  PROC DrawPart60()
    MoveL Offs(pOrigin,354.34,117.20,0.00),v40,z0,tPen\WObj:=wPaper;
    MoveL Offs(pOrigin,355.40,117.41,0.00),v40,z0,tPen\WObj:=wPaper;
    MoveL Offs(pOrigin,355.40,117.41,0.00),v40,z0,tPen\WObj:=wPaper;
    MoveL Offs(pOrigin,357.74,120.39,0.00),v40,z0,tPen\WObj:=wPaper;
    MoveL Offs(pOrigin,361.56,124.00,0.00),v40,z0,tPen\WObj:=wPaper;
    MoveL Offs(pOrigin,364.33,126.12,0.00),v40,z0,tPen\WObj:=wPaper;
    MoveL Offs(pOrigin,368.79,128.89,0.00),v40,fine,tPen\WObj:=wPaper;
    MoveL Offs(pOrigin,368.79,128.89,6.00),v60,z5,tPen\WObj:=wPaper;
    MoveL Offs(pOrigin,367.20,127.37,6.00),vTravel,z5,tPen\WObj:=wPaper;
    MoveL Offs(pOrigin,367.20,127.37,0.00),v60,z0,tPen\WObj:=wPaper;
    MoveL Offs(pOrigin,366.30,128.27,0.00),v40,z0,tPen\WObj:=wPaper;
    MoveL Offs(pOrigin,365.40,127.67,0.00),v40,z0,tPen\WObj:=wPaper;
    MoveL Offs(pOrigin,366.30,126.77,0.00),v40,z0,tPen\WObj:=wPaper;
    MoveL Offs(pOrigin,365.56,126.02,0.00),v40,z0,tPen\WObj:=wPaper;
    MoveL Offs(pOrigin,364.51,127.07,0.00),v40,z0,tPen\WObj:=wPaper;
    MoveL Offs(pOrigin,363.46,126.63,0.00),v40,z0,tPen\WObj:=wPaper;
    MoveL Offs(pOrigin,364.81,125.28,0.00),v40,z0,tPen\WObj:=wPaper;
    MoveL Offs(pOrigin,364.06,124.53,0.00),v40,z0,tPen\WObj:=wPaper;
    MoveL Offs(pOrigin,362.56,126.03,0.00),v40,fine,tPen\WObj:=wPaper;
    MoveL Offs(pOrigin,362.56,126.03,6.00),v60,z5,tPen\WObj:=wPaper;
    MoveL Offs(pOrigin,358.96,129.64,6.00),vTravel,z5,tPen\WObj:=wPaper;
    MoveL Offs(pOrigin,358.96,129.64,0.00),v60,z0,tPen\WObj:=wPaper;
    MoveL Offs(pOrigin,352.19,136.40,0.00),v40,z0,tPen\WObj:=wPaper;
    MoveL Offs(pOrigin,352.71,136.45,0.00),v40,z0,tPen\WObj:=wPaper;
    MoveL Offs(pOrigin,355.71,139.46,0.00),v40,z0,tPen\WObj:=wPaper;
    MoveL Offs(pOrigin,355.40,139.61,0.00),v40,z0,tPen\WObj:=wPaper;
    MoveL Offs(pOrigin,354.12,139.61,0.00),v40,z0,tPen\WObj:=wPaper;
    MoveL Offs(pOrigin,353.77,140.50,0.00),v40,z0,tPen\WObj:=wPaper;
    MoveL Offs(pOrigin,356.62,143.36,0.00),v40,z0,tPen\WObj:=wPaper;
    MoveL Offs(pOrigin,356.46,143.83,0.00),v40,z0,tPen\WObj:=wPaper;
    MoveL Offs(pOrigin,355.19,143.83,0.00),v40,z0,tPen\WObj:=wPaper;
    MoveL Offs(pOrigin,354.68,144.40,0.00),v40,z0,tPen\WObj:=wPaper;
    MoveL Offs(pOrigin,357.68,147.41,0.00),v40,z0,tPen\WObj:=wPaper;
    MoveL Offs(pOrigin,358.00,147.02,0.00),v40,z0,tPen\WObj:=wPaper;
    MoveL Offs(pOrigin,355.60,149.42,0.00),v40,z0,tPen\WObj:=wPaper;
    MoveL Offs(pOrigin,356.46,149.11,0.00),v40,z0,tPen\WObj:=wPaper;
    MoveL Offs(pOrigin,357.52,149.11,0.00),v40,z0,tPen\WObj:=wPaper;
    MoveL Offs(pOrigin,358.14,149.35,0.00),v40,z0,tPen\WObj:=wPaper;
    MoveL Offs(pOrigin,355.13,146.35,0.00),v40,z0,tPen\WObj:=wPaper;
    MoveL Offs(pOrigin,355.61,145.94,0.00),v40,z0,tPen\WObj:=wPaper;
    MoveL Offs(pOrigin,356.89,145.94,0.00),v40,z0,tPen\WObj:=wPaper;
    MoveL Offs(pOrigin,357.23,145.46,0.00),v40,z0,tPen\WObj:=wPaper;
    MoveL Offs(pOrigin,354.22,142.45,0.00),v40,z0,tPen\WObj:=wPaper;
    MoveL Offs(pOrigin,353.82,142.24,0.00),v40,z0,tPen\WObj:=wPaper;
    MoveL Offs(pOrigin,356.38,139.68,0.00),v40,fine,tPen\WObj:=wPaper;
    MoveL Offs(pOrigin,356.38,139.68,6.00),v60,z5,tPen\WObj:=wPaper;
    MoveL Offs(pOrigin,356.08,138.49,6.00),vTravel,z5,tPen\WObj:=wPaper;
    MoveL Offs(pOrigin,356.08,138.49,0.00),v60,z0,tPen\WObj:=wPaper;
    MoveL Offs(pOrigin,353.53,141.04,0.00),v40,z0,tPen\WObj:=wPaper;
    MoveL Offs(pOrigin,354.34,140.66,0.00),v40,z0,tPen\WObj:=wPaper;
    MoveL Offs(pOrigin,355.61,140.66,0.00),v40,z0,tPen\WObj:=wPaper;
    MoveL Offs(pOrigin,356.17,141.41,0.00),v40,z0,tPen\WObj:=wPaper;
    MoveL Offs(pOrigin,353.16,138.40,0.00),v40,z0,tPen\WObj:=wPaper;
    MoveL Offs(pOrigin,352.94,138.64,0.00),v40,z0,tPen\WObj:=wPaper;
    MoveL Offs(pOrigin,360.30,131.28,0.00),v40,z0,tPen\WObj:=wPaper;
    MoveL Offs(pOrigin,360.08,132.22,0.00),v40,z0,tPen\WObj:=wPaper;
    MoveL Offs(pOrigin,358.16,132.22,0.00),v40,fine,tPen\WObj:=wPaper;
    MoveL Offs(pOrigin,358.16,132.22,6.00),v60,z5,tPen\WObj:=wPaper;
    MoveL Offs(pOrigin,359.23,131.44,6.00),vTravel,z5,tPen\WObj:=wPaper;
    MoveL Offs(pOrigin,359.23,131.44,0.00),v60,z0,tPen\WObj:=wPaper;
    MoveL Offs(pOrigin,359.65,131.86,0.00),v40,z0,tPen\WObj:=wPaper;
    MoveL Offs(pOrigin,359.23,131.44,0.00),v40,z0,tPen\WObj:=wPaper;
    MoveL Offs(pOrigin,359.22,131.16,0.00),v40,z0,tPen\WObj:=wPaper;
    MoveL Offs(pOrigin,357.31,131.16,0.00),v40,fine,tPen\WObj:=wPaper;
    MoveL Offs(pOrigin,357.31,131.16,6.00),v60,z5,tPen\WObj:=wPaper;
    MoveL Offs(pOrigin,358.38,130.38,6.00),vTravel,z5,tPen\WObj:=wPaper;
    MoveL Offs(pOrigin,358.38,130.38,0.00),v60,z0,tPen\WObj:=wPaper;
    MoveL Offs(pOrigin,358.80,130.80,0.00),v40,z0,tPen\WObj:=wPaper;
    MoveL Offs(pOrigin,358.38,130.38,0.00),v40,z0,tPen\WObj:=wPaper;
    MoveL Offs(pOrigin,358.38,130.10,0.00),v40,z0,tPen\WObj:=wPaper;
    MoveL Offs(pOrigin,356.46,130.10,0.00),v40,fine,tPen\WObj:=wPaper;
    MoveL Offs(pOrigin,356.46,130.10,6.00),v60,z5,tPen\WObj:=wPaper;
    MoveL Offs(pOrigin,357.52,129.31,6.00),vTravel,z5,tPen\WObj:=wPaper;
    MoveL Offs(pOrigin,357.52,129.31,0.00),v60,z0,tPen\WObj:=wPaper;
    MoveL Offs(pOrigin,357.95,129.74,0.00),v40,z0,tPen\WObj:=wPaper;
    MoveL Offs(pOrigin,357.52,129.31,0.00),v40,z0,tPen\WObj:=wPaper;
    MoveL Offs(pOrigin,357.52,129.05,0.00),v40,z0,tPen\WObj:=wPaper;
    MoveL Offs(pOrigin,355.61,129.05,0.00),v40,z0,tPen\WObj:=wPaper;
    MoveL Offs(pOrigin,355.61,128.68,0.00),v40,z0,tPen\WObj:=wPaper;
    MoveL Offs(pOrigin,356.04,129.31,0.00),v40,z0,tPen\WObj:=wPaper;
    MoveL Offs(pOrigin,355.61,128.68,0.00),v40,fine,tPen\WObj:=wPaper;
    MoveL Offs(pOrigin,355.61,128.68,6.00),v60,z5,tPen\WObj:=wPaper;
    MoveL Offs(pOrigin,356.67,128.04,6.00),vTravel,z5,tPen\WObj:=wPaper;
    MoveL Offs(pOrigin,356.67,128.04,0.00),v60,z0,tPen\WObj:=wPaper;
    MoveL Offs(pOrigin,357.31,128.89,0.00),v40,z0,tPen\WObj:=wPaper;
    MoveL Offs(pOrigin,356.67,128.04,0.00),v40,z0,tPen\WObj:=wPaper;
    MoveL Offs(pOrigin,356.67,127.99,0.00),v40,z0,tPen\WObj:=wPaper;
    MoveL Offs(pOrigin,351.58,127.99,0.00),v40,z0,tPen\WObj:=wPaper;
    MoveL Offs(pOrigin,351.66,126.98,0.00),v40,z0,tPen\WObj:=wPaper;
    MoveL Offs(pOrigin,351.66,119.32,0.00),v40,z0,tPen\WObj:=wPaper;
    MoveL Offs(pOrigin,352.42,119.54,0.00),v40,z0,tPen\WObj:=wPaper;
    MoveL Offs(pOrigin,349.88,119.54,0.00),v40,z0,tPen\WObj:=wPaper;
    MoveL Offs(pOrigin,349.36,119.67,0.00),v40,z0,tPen\WObj:=wPaper;
    MoveL Offs(pOrigin,356.42,126.73,0.00),v40,z0,tPen\WObj:=wPaper;
    MoveL Offs(pOrigin,356.04,126.94,0.00),v40,z0,tPen\WObj:=wPaper;
    MoveL Offs(pOrigin,351.36,126.94,0.00),v40,z0,tPen\WObj:=wPaper;
    MoveL Offs(pOrigin,350.88,127.16,0.00),v40,z0,tPen\WObj:=wPaper;
    MoveL Offs(pOrigin,360.50,136.78,0.00),v40,fine,tPen\WObj:=wPaper;
    MoveL Offs(pOrigin,360.50,136.78,6.00),v60,z5,tPen\WObj:=wPaper;
    MoveL Offs(pOrigin,360.50,138.24,6.00),vTravel,z5,tPen\WObj:=wPaper;
    MoveL Offs(pOrigin,360.50,138.24,0.00),v60,z0,tPen\WObj:=wPaper;
    MoveL Offs(pOrigin,360.92,138.24,0.00),v40,z0,tPen\WObj:=wPaper;
    MoveL Offs(pOrigin,361.99,139.30,0.00),v40,z0,tPen\WObj:=wPaper;
    MoveL Offs(pOrigin,362.20,140.15,0.00),v40,z0,tPen\WObj:=wPaper;
    MoveL Offs(pOrigin,362.20,140.15,0.00),v40,z0,tPen\WObj:=wPaper;
    MoveL Offs(pOrigin,363.26,141.21,0.00),v40,z0,tPen\WObj:=wPaper;
    MoveL Offs(pOrigin,363.26,141.21,0.00),v40,z0,tPen\WObj:=wPaper;
    MoveL Offs(pOrigin,363.33,141.85,0.00),v40,z0,tPen\WObj:=wPaper;
    MoveL Offs(pOrigin,365.17,143.62,0.00),v40,z0,tPen\WObj:=wPaper;
    MoveL Offs(pOrigin,365.81,143.76,0.00),v40,fine,tPen\WObj:=wPaper;
    MoveL Offs(pOrigin,365.81,143.76,6.00),v60,z5,tPen\WObj:=wPaper;
    MoveL Offs(pOrigin,366.70,142.80,6.00),vTravel,z5,tPen\WObj:=wPaper;
    MoveL Offs(pOrigin,366.70,142.80,0.00),v60,z0,tPen\WObj:=wPaper;
    MoveL Offs(pOrigin,362.50,147.00,0.00),v40,z0,tPen\WObj:=wPaper;
    MoveL Offs(pOrigin,362.92,146.67,0.00),v40,z0,tPen\WObj:=wPaper;
    MoveL Offs(pOrigin,376.15,159.90,0.00),v40,z0,tPen\WObj:=wPaper;
    MoveL Offs(pOrigin,376.01,160.12,0.00),v40,z0,tPen\WObj:=wPaper;
    MoveL Offs(pOrigin,376.65,160.76,0.00),v40,z0,tPen\WObj:=wPaper;
    MoveL Offs(pOrigin,376.01,160.12,0.00),v40,z0,tPen\WObj:=wPaper;
    MoveL Offs(pOrigin,376.22,160.73,0.00),v40,z0,tPen\WObj:=wPaper;
  ENDPROC

  PROC DrawPart61()
    MoveL Offs(pOrigin,374.95,160.73,0.00),v40,z0,tPen\WObj:=wPaper;
    MoveL Offs(pOrigin,375.38,159.67,0.00),v40,z0,tPen\WObj:=wPaper;
    MoveL Offs(pOrigin,374.10,159.67,0.00),v40,z0,tPen\WObj:=wPaper;
    MoveL Offs(pOrigin,373.30,160.04,0.00),v40,z0,tPen\WObj:=wPaper;
    MoveL Offs(pOrigin,381.72,168.45,0.00),v40,z0,tPen\WObj:=wPaper;
    MoveL Offs(pOrigin,381.91,167.92,0.00),v40,z0,tPen\WObj:=wPaper;
    MoveL Offs(pOrigin,379.35,170.47,0.00),v40,z0,tPen\WObj:=wPaper;
    MoveL Offs(pOrigin,379.78,170.99,0.00),v40,z0,tPen\WObj:=wPaper;
    MoveL Offs(pOrigin,381.58,172.79,0.00),v40,z0,tPen\WObj:=wPaper;
    MoveL Offs(pOrigin,381.11,172.34,0.00),v40,z0,tPen\WObj:=wPaper;
    MoveL Offs(pOrigin,380.05,172.34,0.00),v40,z0,tPen\WObj:=wPaper;
    MoveL Offs(pOrigin,379.48,172.19,0.00),v40,z0,tPen\WObj:=wPaper;
    MoveL Offs(pOrigin,381.13,173.84,0.00),v40,z0,tPen\WObj:=wPaper;
    MoveL Offs(pOrigin,380.90,173.40,0.00),v40,z0,tPen\WObj:=wPaper;
    MoveL Offs(pOrigin,379.62,173.40,0.00),v40,z0,tPen\WObj:=wPaper;
    MoveL Offs(pOrigin,379.18,173.39,0.00),v40,z0,tPen\WObj:=wPaper;
    MoveL Offs(pOrigin,380.69,174.89,0.00),v40,z0,tPen\WObj:=wPaper;
    MoveL Offs(pOrigin,380.48,174.46,0.00),v40,z0,tPen\WObj:=wPaper;
    MoveL Offs(pOrigin,379.20,174.46,0.00),v40,z0,tPen\WObj:=wPaper;
    MoveL Offs(pOrigin,378.74,174.43,0.00),v40,z0,tPen\WObj:=wPaper;
    MoveL Offs(pOrigin,380.24,175.94,0.00),v40,z0,tPen\WObj:=wPaper;
    MoveL Offs(pOrigin,380.05,175.51,0.00),v40,z0,tPen\WObj:=wPaper;
    MoveL Offs(pOrigin,378.78,175.51,0.00),v40,z0,tPen\WObj:=wPaper;
    MoveL Offs(pOrigin,378.29,175.48,0.00),v40,z0,tPen\WObj:=wPaper;
    MoveL Offs(pOrigin,379.94,177.13,0.00),v40,z0,tPen\WObj:=wPaper;
    MoveL Offs(pOrigin,379.62,176.57,0.00),v40,z0,tPen\WObj:=wPaper;
    MoveL Offs(pOrigin,378.56,176.57,0.00),v40,z0,tPen\WObj:=wPaper;
    MoveL Offs(pOrigin,377.85,176.53,0.00),v40,z0,tPen\WObj:=wPaper;
    MoveL Offs(pOrigin,379.65,178.33,0.00),v40,z0,tPen\WObj:=wPaper;
    MoveL Offs(pOrigin,380.08,178.71,0.00),v40,z0,tPen\WObj:=wPaper;
    MoveL Offs(pOrigin,374.22,184.57,0.00),v40,z0,tPen\WObj:=wPaper;
    MoveL Offs(pOrigin,373.62,183.67,0.00),v40,z0,tPen\WObj:=wPaper;
    MoveL Offs(pOrigin,375.12,182.17,0.00),v40,z0,tPen\WObj:=wPaper;
    MoveL Offs(pOrigin,374.68,181.12,0.00),v40,z0,tPen\WObj:=wPaper;
    MoveL Offs(pOrigin,373.17,182.62,0.00),v40,z0,tPen\WObj:=wPaper;
    MoveL Offs(pOrigin,372.73,181.58,0.00),v40,z0,tPen\WObj:=wPaper;
    MoveL Offs(pOrigin,374.08,180.22,0.00),v40,z0,tPen\WObj:=wPaper;
    MoveL Offs(pOrigin,373.63,179.18,0.00),v40,z0,tPen\WObj:=wPaper;
    MoveL Offs(pOrigin,372.13,180.68,0.00),v40,z0,tPen\WObj:=wPaper;
    MoveL Offs(pOrigin,371.68,179.63,0.00),v40,z0,tPen\WObj:=wPaper;
    MoveL Offs(pOrigin,373.19,178.13,0.00),v40,z0,tPen\WObj:=wPaper;
    MoveL Offs(pOrigin,372.59,177.23,0.00),v40,z0,tPen\WObj:=wPaper;
    MoveL Offs(pOrigin,371.24,178.59,0.00),v40,z0,tPen\WObj:=wPaper;
    MoveL Offs(pOrigin,370.79,177.54,0.00),v40,z0,tPen\WObj:=wPaper;
    MoveL Offs(pOrigin,372.14,176.19,0.00),v40,z0,tPen\WObj:=wPaper;
    MoveL Offs(pOrigin,371.70,175.14,0.00),v40,z0,tPen\WObj:=wPaper;
    MoveL Offs(pOrigin,370.65,176.19,0.00),v40,z0,tPen\WObj:=wPaper;
    MoveL Offs(pOrigin,370.20,175.14,0.00),v40,z0,tPen\WObj:=wPaper;
    MoveL Offs(pOrigin,371.10,174.24,0.00),v40,fine,tPen\WObj:=wPaper;
    MoveL Offs(pOrigin,371.10,174.24,6.00),v60,z5,tPen\WObj:=wPaper;
    MoveL Offs(pOrigin,369.85,171.39,6.00),vTravel,z5,tPen\WObj:=wPaper;
    MoveL Offs(pOrigin,369.85,171.39,0.00),v60,z0,tPen\WObj:=wPaper;
    MoveL Offs(pOrigin,369.85,172.24,0.00),v40,z0,tPen\WObj:=wPaper;
    MoveL Offs(pOrigin,371.69,177.12,0.00),v40,z0,tPen\WObj:=wPaper;
    MoveL Offs(pOrigin,375.38,184.99,0.00),v40,z0,tPen\WObj:=wPaper;
    MoveL Offs(pOrigin,375.38,184.99,0.00),v40,z0,tPen\WObj:=wPaper;
    MoveL Offs(pOrigin,375.59,186.69,0.00),v40,z0,tPen\WObj:=wPaper;
    MoveL Offs(pOrigin,374.95,187.75,0.00),v40,z0,tPen\WObj:=wPaper;
    MoveL Offs(pOrigin,374.29,187.90,0.00),v40,z0,tPen\WObj:=wPaper;
    MoveL Offs(pOrigin,375.64,189.25,0.00),v40,z0,tPen\WObj:=wPaper;
    MoveL Offs(pOrigin,374.74,189.24,0.00),v40,z0,tPen\WObj:=wPaper;
    MoveL Offs(pOrigin,369.64,189.24,0.00),v40,z0,tPen\WObj:=wPaper;
    MoveL Offs(pOrigin,368.60,189.68,0.00),v40,z0,tPen\WObj:=wPaper;
    MoveL Offs(pOrigin,370.25,191.34,0.00),v40,z0,tPen\WObj:=wPaper;
    MoveL Offs(pOrigin,369.85,191.92,0.00),v40,z0,tPen\WObj:=wPaper;
    MoveL Offs(pOrigin,379.32,182.46,0.00),v40,z0,tPen\WObj:=wPaper;
    MoveL Offs(pOrigin,379.06,182.22,0.00),v40,z0,tPen\WObj:=wPaper;
    MoveL Offs(pOrigin,377.26,180.42,0.00),v40,z0,tPen\WObj:=wPaper;
    MoveL Offs(pOrigin,376.63,180.67,0.00),v40,z0,tPen\WObj:=wPaper;
    MoveL Offs(pOrigin,380.68,176.61,0.00),v40,fine,tPen\WObj:=wPaper;
    MoveL Offs(pOrigin,380.68,176.61,6.00),v60,z5,tPen\WObj:=wPaper;
    MoveL Offs(pOrigin,379.20,177.62,6.00),vTravel,z5,tPen\WObj:=wPaper;
    MoveL Offs(pOrigin,379.20,177.62,0.00),v60,z0,tPen\WObj:=wPaper;
    MoveL Offs(pOrigin,378.14,177.62,0.00),v40,z0,tPen\WObj:=wPaper;
    MoveL Offs(pOrigin,377.70,177.88,0.00),v40,z0,tPen\WObj:=wPaper;
    MoveL Offs(pOrigin,379.35,179.53,0.00),v40,z0,tPen\WObj:=wPaper;
    MoveL Offs(pOrigin,378.99,178.68,0.00),v40,z0,tPen\WObj:=wPaper;
    MoveL Offs(pOrigin,377.92,178.68,0.00),v40,z0,tPen\WObj:=wPaper;
    MoveL Offs(pOrigin,377.40,179.07,0.00),v40,z0,tPen\WObj:=wPaper;
    MoveL Offs(pOrigin,379.21,180.88,0.00),v40,z0,tPen\WObj:=wPaper;
    MoveL Offs(pOrigin,379.77,180.51,0.00),v40,z0,tPen\WObj:=wPaper;
    MoveL Offs(pOrigin,374.51,185.77,0.00),v40,z0,tPen\WObj:=wPaper;
    MoveL Offs(pOrigin,375.03,185.66,0.00),v40,z0,tPen\WObj:=wPaper;
    MoveL Offs(pOrigin,377.13,187.76,0.00),v40,z0,tPen\WObj:=wPaper;
    MoveL Offs(pOrigin,377.08,187.11,0.00),v40,z0,tPen\WObj:=wPaper;
    MoveL Offs(pOrigin,376.65,187.75,0.00),v40,z0,tPen\WObj:=wPaper;
    MoveL Offs(pOrigin,377.08,187.11,0.00),v40,z0,tPen\WObj:=wPaper;
    MoveL Offs(pOrigin,376.86,187.13,0.00),v40,z0,tPen\WObj:=wPaper;
    MoveL Offs(pOrigin,375.38,187.13,0.00),v40,z0,tPen\WObj:=wPaper;
    MoveL Offs(pOrigin,375.38,186.90,0.00),v40,z0,tPen\WObj:=wPaper;
    MoveL Offs(pOrigin,375.16,187.32,0.00),v40,z0,tPen\WObj:=wPaper;
    MoveL Offs(pOrigin,375.38,186.90,0.00),v40,z0,tPen\WObj:=wPaper;
    MoveL Offs(pOrigin,374.88,187.01,0.00),v40,z0,tPen\WObj:=wPaper;
    MoveL Offs(pOrigin,376.38,188.51,0.00),v40,z0,tPen\WObj:=wPaper;
    MoveL Offs(pOrigin,376.44,188.18,0.00),v40,z0,tPen\WObj:=wPaper;
    MoveL Offs(pOrigin,375.38,189.24,0.00),v40,z0,tPen\WObj:=wPaper;
    MoveL Offs(pOrigin,376.44,188.18,0.00),v40,z0,tPen\WObj:=wPaper;
    MoveL Offs(pOrigin,375.80,188.18,0.00),v40,z0,tPen\WObj:=wPaper;
    MoveL Offs(pOrigin,374.31,188.18,0.00),v40,z0,tPen\WObj:=wPaper;
    MoveL Offs(pOrigin,374.10,188.18,0.00),v40,z0,tPen\WObj:=wPaper;
    MoveL Offs(pOrigin,374.38,188.03,0.00),v40,z0,tPen\WObj:=wPaper;
    MoveL Offs(pOrigin,372.40,189.02,0.00),v40,z0,tPen\WObj:=wPaper;
    MoveL Offs(pOrigin,371.34,189.02,0.00),v40,z0,tPen\WObj:=wPaper;
    MoveL Offs(pOrigin,370.27,188.18,0.00),v40,z0,tPen\WObj:=wPaper;
    MoveL Offs(pOrigin,368.43,184.99,0.00),v40,z0,tPen\WObj:=wPaper;
    MoveL Offs(pOrigin,365.95,178.61,0.00),v40,z0,tPen\WObj:=wPaper;
    MoveL Offs(pOrigin,362.62,167.77,0.00),v40,z0,tPen\WObj:=wPaper;
    MoveL Offs(pOrigin,357.74,149.50,0.00),v40,z0,tPen\WObj:=wPaper;
    MoveL Offs(pOrigin,353.70,131.86,0.00),v40,z0,tPen\WObj:=wPaper;
    MoveL Offs(pOrigin,354.12,130.80,0.00),v40,z0,tPen\WObj:=wPaper;
    MoveL Offs(pOrigin,353.91,130.38,0.00),v40,z0,tPen\WObj:=wPaper;
    MoveL Offs(pOrigin,354.12,130.80,0.00),v40,z0,tPen\WObj:=wPaper;
    MoveL Offs(pOrigin,353.91,130.38,0.00),v40,z0,tPen\WObj:=wPaper;
    MoveL Offs(pOrigin,354.55,130.10,0.00),v40,z0,tPen\WObj:=wPaper;
    MoveL Offs(pOrigin,352.00,130.10,0.00),v40,z0,tPen\WObj:=wPaper;
    MoveL Offs(pOrigin,351.49,130.76,0.00),v40,z0,tPen\WObj:=wPaper;
    MoveL Offs(pOrigin,354.95,134.21,0.00),v40,z0,tPen\WObj:=wPaper;
    MoveL Offs(pOrigin,354.34,134.33,0.00),v40,z0,tPen\WObj:=wPaper;
    MoveL Offs(pOrigin,352.85,134.33,0.00),v40,z0,tPen\WObj:=wPaper;
    MoveL Offs(pOrigin,352.25,134.51,0.00),v40,z0,tPen\WObj:=wPaper;
  ENDPROC

  PROC DrawPart62()
    MoveL Offs(pOrigin,355.41,137.66,0.00),v40,z0,tPen\WObj:=wPaper;
    MoveL Offs(pOrigin,355.64,137.44,0.00),v40,z0,tPen\WObj:=wPaper;
    MoveL Offs(pOrigin,353.08,139.99,0.00),v40,fine,tPen\WObj:=wPaper;
    MoveL Offs(pOrigin,353.08,139.99,6.00),v60,z5,tPen\WObj:=wPaper;
    MoveL Offs(pOrigin,353.91,138.55,6.00),vTravel,z5,tPen\WObj:=wPaper;
    MoveL Offs(pOrigin,353.91,138.55,0.00),v60,z0,tPen\WObj:=wPaper;
    MoveL Offs(pOrigin,355.19,138.55,0.00),v40,z0,tPen\WObj:=wPaper;
    MoveL Offs(pOrigin,354.98,137.50,0.00),v40,z0,tPen\WObj:=wPaper;
    MoveL Offs(pOrigin,353.70,137.50,0.00),v40,z0,tPen\WObj:=wPaper;
    MoveL Offs(pOrigin,353.49,136.44,0.00),v40,z0,tPen\WObj:=wPaper;
    MoveL Offs(pOrigin,354.76,136.44,0.00),v40,z0,tPen\WObj:=wPaper;
    MoveL Offs(pOrigin,354.95,135.71,0.00),v40,z0,tPen\WObj:=wPaper;
    MoveL Offs(pOrigin,351.95,132.71,0.00),v40,z0,tPen\WObj:=wPaper;
    MoveL Offs(pOrigin,351.46,132.66,0.00),v40,z0,tPen\WObj:=wPaper;
    MoveL Offs(pOrigin,357.02,127.10,0.00),v40,z0,tPen\WObj:=wPaper;
    MoveL Offs(pOrigin,356.25,127.40,0.00),v40,z0,tPen\WObj:=wPaper;
    MoveL Offs(pOrigin,356.46,127.82,0.00),v40,z0,tPen\WObj:=wPaper;
    MoveL Offs(pOrigin,356.25,127.40,0.00),v40,fine,tPen\WObj:=wPaper;
    MoveL Offs(pOrigin,356.25,127.40,6.00),v60,z5,tPen\WObj:=wPaper;
    MoveL Offs(pOrigin,355.61,126.34,6.00),vTravel,z5,tPen\WObj:=wPaper;
    MoveL Offs(pOrigin,355.61,126.34,0.00),v60,z0,tPen\WObj:=wPaper;
    MoveL Offs(pOrigin,355.83,126.76,0.00),v40,z0,tPen\WObj:=wPaper;
    MoveL Offs(pOrigin,355.61,126.34,0.00),v40,z0,tPen\WObj:=wPaper;
    MoveL Offs(pOrigin,355.40,125.88,0.00),v40,z0,tPen\WObj:=wPaper;
    MoveL Offs(pOrigin,351.15,125.88,0.00),v40,fine,tPen\WObj:=wPaper;
    MoveL Offs(pOrigin,351.15,125.88,6.00),v60,z5,tPen\WObj:=wPaper;
    MoveL Offs(pOrigin,350.13,126.52,6.00),vTravel,z5,tPen\WObj:=wPaper;
    MoveL Offs(pOrigin,350.13,126.52,0.00),v60,z0,tPen\WObj:=wPaper;
    MoveL Offs(pOrigin,354.48,122.16,0.00),v40,z0,tPen\WObj:=wPaper;
    MoveL Offs(pOrigin,353.70,122.71,0.00),v40,z0,tPen\WObj:=wPaper;
    MoveL Offs(pOrigin,350.51,122.71,0.00),v40,z0,tPen\WObj:=wPaper;
    MoveL Offs(pOrigin,350.61,122.09,0.00),v40,z0,tPen\WObj:=wPaper;
    MoveL Offs(pOrigin,350.61,116.14,0.00),v40,z0,tPen\WObj:=wPaper;
    MoveL Offs(pOrigin,351.36,116.38,0.00),v40,z0,tPen\WObj:=wPaper;
    MoveL Offs(pOrigin,349.24,116.38,0.00),v40,z0,tPen\WObj:=wPaper;
    MoveL Offs(pOrigin,349.55,116.56,0.00),v40,z0,tPen\WObj:=wPaper;
    MoveL Offs(pOrigin,349.55,105.30,0.00),v40,z0,tPen\WObj:=wPaper;
    MoveL Offs(pOrigin,349.88,104.76,0.00),v40,z0,tPen\WObj:=wPaper;
    MoveL Offs(pOrigin,346.05,104.76,0.00),v40,z0,tPen\WObj:=wPaper;
    MoveL Offs(pOrigin,345.10,104.66,0.00),v40,z0,tPen\WObj:=wPaper;
    MoveL Offs(pOrigin,350.36,99.41,0.00),v40,z0,tPen\WObj:=wPaper;
    MoveL Offs(pOrigin,349.91,98.36,0.00),v40,z0,tPen\WObj:=wPaper;
    MoveL Offs(pOrigin,344.80,103.47,0.00),v40,z0,tPen\WObj:=wPaper;
    MoveL Offs(pOrigin,344.81,103.18,0.00),v40,z0,tPen\WObj:=wPaper;
    MoveL Offs(pOrigin,354.73,113.09,0.00),v40,z0,tPen\WObj:=wPaper;
    MoveL Offs(pOrigin,355.41,113.77,0.00),v40,z0,tPen\WObj:=wPaper;
    MoveL Offs(pOrigin,357.51,111.67,0.00),v40,z0,tPen\WObj:=wPaper;
    MoveL Offs(pOrigin,356.67,112.15,0.00),v40,z0,tPen\WObj:=wPaper;
    MoveL Offs(pOrigin,354.98,112.15,0.00),v40,z0,tPen\WObj:=wPaper;
    MoveL Offs(pOrigin,355.40,111.10,0.00),v40,z0,tPen\WObj:=wPaper;
    MoveL Offs(pOrigin,353.06,111.10,0.00),v40,fine,tPen\WObj:=wPaper;
    MoveL Offs(pOrigin,353.06,111.10,6.00),v60,z5,tPen\WObj:=wPaper;
    MoveL Offs(pOrigin,352.00,112.15,6.00),vTravel,z5,tPen\WObj:=wPaper;
    MoveL Offs(pOrigin,352.00,112.15,0.00),v60,z0,tPen\WObj:=wPaper;
    MoveL Offs(pOrigin,348.17,112.15,0.00),v40,z0,tPen\WObj:=wPaper;
    MoveL Offs(pOrigin,348.49,112.10,0.00),v40,z0,tPen\WObj:=wPaper;
    MoveL Offs(pOrigin,348.49,95.31,0.00),v40,z0,tPen\WObj:=wPaper;
    MoveL Offs(pOrigin,347.96,95.26,0.00),v40,z0,tPen\WObj:=wPaper;
    MoveL Offs(pOrigin,349.88,95.26,0.00),v40,z0,tPen\WObj:=wPaper;
    MoveL Offs(pOrigin,349.55,94.89,0.00),v40,z0,tPen\WObj:=wPaper;
    MoveL Offs(pOrigin,349.55,89.58,0.00),v40,z0,tPen\WObj:=wPaper;
    MoveL Offs(pOrigin,348.60,89.98,0.00),v40,z0,tPen\WObj:=wPaper;
    MoveL Offs(pOrigin,353.28,89.98,0.00),v40,z0,tPen\WObj:=wPaper;
    MoveL Offs(pOrigin,353.61,89.57,0.00),v40,z0,tPen\WObj:=wPaper;
    MoveL Offs(pOrigin,347.45,83.41,0.00),v40,z0,tPen\WObj:=wPaper;
    MoveL Offs(pOrigin,346.96,83.39,0.00),v40,z0,tPen\WObj:=wPaper;
    MoveL Offs(pOrigin,349.97,80.38,0.00),v40,fine,tPen\WObj:=wPaper;
    MoveL Offs(pOrigin,349.97,80.38,6.00),v60,z5,tPen\WObj:=wPaper;
    MoveL Offs(pOrigin,349.82,79.03,6.00),vTravel,z5,tPen\WObj:=wPaper;
    MoveL Offs(pOrigin,349.82,79.03,0.00),v60,z0,tPen\WObj:=wPaper;
    MoveL Offs(pOrigin,346.82,82.04,0.00),v40,z0,tPen\WObj:=wPaper;
    MoveL Offs(pOrigin,347.30,81.76,0.00),v40,z0,tPen\WObj:=wPaper;
    MoveL Offs(pOrigin,353.61,88.07,0.00),v40,z0,tPen\WObj:=wPaper;
    MoveL Offs(pOrigin,353.28,87.86,0.00),v40,z0,tPen\WObj:=wPaper;
    MoveL Offs(pOrigin,351.36,87.86,0.00),v40,z0,tPen\WObj:=wPaper;
    MoveL Offs(pOrigin,351.66,88.30,0.00),v40,z0,tPen\WObj:=wPaper;
    MoveL Offs(pOrigin,351.66,91.91,0.00),v40,z0,tPen\WObj:=wPaper;
    MoveL Offs(pOrigin,352.42,91.91,0.00),v40,z0,tPen\WObj:=wPaper;
    MoveL Offs(pOrigin,352.00,92.12,0.00),v40,z0,tPen\WObj:=wPaper;
    MoveL Offs(pOrigin,349.38,96.38,0.00),v40,z0,tPen\WObj:=wPaper;
    MoveL Offs(pOrigin,349.02,97.44,0.00),v40,z0,tPen\WObj:=wPaper;
    MoveL Offs(pOrigin,349.17,99.35,0.00),v40,z0,tPen\WObj:=wPaper;
    MoveL Offs(pOrigin,350.73,101.69,0.00),v40,z0,tPen\WObj:=wPaper;
    MoveL Offs(pOrigin,357.10,107.78,0.00),v40,z0,tPen\WObj:=wPaper;
    MoveL Offs(pOrigin,358.30,108.35,0.00),v40,z0,tPen\WObj:=wPaper;
    MoveL Offs(pOrigin,358.80,109.27,0.00),v40,z0,tPen\WObj:=wPaper;
    MoveL Offs(pOrigin,366.02,113.66,0.00),v40,z0,tPen\WObj:=wPaper;
    MoveL Offs(pOrigin,377.29,119.40,0.00),v40,z0,tPen\WObj:=wPaper;
    MoveL Offs(pOrigin,384.94,122.58,0.00),v40,z0,tPen\WObj:=wPaper;
    MoveL Offs(pOrigin,387.49,123.36,0.00),v40,z0,tPen\WObj:=wPaper;
    MoveL Offs(pOrigin,388.55,123.36,0.00),v40,fine,tPen\WObj:=wPaper;
    MoveL Offs(pOrigin,388.55,123.36,6.00),v60,z5,tPen\WObj:=wPaper;
    MoveL Offs(pOrigin,387.58,124.91,6.00),vTravel,z5,tPen\WObj:=wPaper;
    MoveL Offs(pOrigin,387.58,124.91,0.00),v60,z0,tPen\WObj:=wPaper;
    MoveL Offs(pOrigin,385.33,127.16,0.00),v40,fine,tPen\WObj:=wPaper;
    MoveL Offs(pOrigin,385.33,127.16,6.00),v60,z5,tPen\WObj:=wPaper;
    MoveL Offs(pOrigin,384.51,125.70,6.00),vTravel,z5,tPen\WObj:=wPaper;
    MoveL Offs(pOrigin,384.51,125.70,0.00),v60,z0,tPen\WObj:=wPaper;
    MoveL Offs(pOrigin,385.36,125.49,0.00),v40,z0,tPen\WObj:=wPaper;
    MoveL Offs(pOrigin,392.16,126.97,0.00),v40,z0,tPen\WObj:=wPaper;
    MoveL Offs(pOrigin,393.65,126.97,0.00),v40,z0,tPen\WObj:=wPaper;
    MoveL Offs(pOrigin,395.00,126.12,0.00),v40,z0,tPen\WObj:=wPaper;
    MoveL Offs(pOrigin,395.35,125.06,0.00),v40,z0,tPen\WObj:=wPaper;
    MoveL Offs(pOrigin,395.14,118.47,0.00),v40,z0,tPen\WObj:=wPaper;
    MoveL Offs(pOrigin,396.06,116.21,0.00),v40,z0,tPen\WObj:=wPaper;
    MoveL Offs(pOrigin,398.61,112.53,0.00),v40,z0,tPen\WObj:=wPaper;
    MoveL Offs(pOrigin,400.02,108.28,0.00),v40,z0,tPen\WObj:=wPaper;
    MoveL Offs(pOrigin,399.95,107.64,0.00),v40,z0,tPen\WObj:=wPaper;
    MoveL Offs(pOrigin,399.17,107.71,0.00),v40,z0,tPen\WObj:=wPaper;
    MoveL Offs(pOrigin,393.86,110.68,0.00),v40,z0,tPen\WObj:=wPaper;
    MoveL Offs(pOrigin,391.10,111.46,0.00),v40,z0,tPen\WObj:=wPaper;
    MoveL Offs(pOrigin,391.10,111.46,0.00),v40,z0,tPen\WObj:=wPaper;
    MoveL Offs(pOrigin,391.74,110.54,0.00),v40,z0,tPen\WObj:=wPaper;
    MoveL Offs(pOrigin,395.35,108.77,0.00),v40,z0,tPen\WObj:=wPaper;
    MoveL Offs(pOrigin,398.40,106.65,0.00),v40,z0,tPen\WObj:=wPaper;
    MoveL Offs(pOrigin,398.11,106.79,0.00),v40,z0,tPen\WObj:=wPaper;
    MoveL Offs(pOrigin,398.33,106.87,0.00),v40,z0,tPen\WObj:=wPaper;
    MoveL Offs(pOrigin,401.94,106.87,0.00),v40,z0,tPen\WObj:=wPaper;
    MoveL Offs(pOrigin,402.35,106.95,0.00),v40,z0,tPen\WObj:=wPaper;
    MoveL Offs(pOrigin,400.10,104.69,0.00),v40,z0,tPen\WObj:=wPaper;
  ENDPROC

  PROC DrawPart63()
    MoveL Offs(pOrigin,400.24,105.09,0.00),v40,z0,tPen\WObj:=wPaper;
    MoveL Offs(pOrigin,400.02,105.51,0.00),v40,z0,tPen\WObj:=wPaper;
    MoveL Offs(pOrigin,400.24,105.09,0.00),v40,z0,tPen\WObj:=wPaper;
    MoveL Offs(pOrigin,400.66,104.88,0.00),v40,z0,tPen\WObj:=wPaper;
    MoveL Offs(pOrigin,400.88,104.45,0.00),v40,z0,tPen\WObj:=wPaper;
    MoveL Offs(pOrigin,400.66,104.88,0.00),v40,z0,tPen\WObj:=wPaper;
    MoveL Offs(pOrigin,400.66,104.76,0.00),v40,z0,tPen\WObj:=wPaper;
    MoveL Offs(pOrigin,402.79,104.76,0.00),v40,z0,tPen\WObj:=wPaper;
    MoveL Offs(pOrigin,403.39,105.00,0.00),v40,z0,tPen\WObj:=wPaper;
    MoveL Offs(pOrigin,401.59,103.20,0.00),v40,z0,tPen\WObj:=wPaper;
    MoveL Offs(pOrigin,401.72,103.70,0.00),v40,z0,tPen\WObj:=wPaper;
    MoveL Offs(pOrigin,403.64,103.70,0.00),v40,z0,tPen\WObj:=wPaper;
    MoveL Offs(pOrigin,403.85,103.60,0.00),v40,z0,tPen\WObj:=wPaper;
    MoveL Offs(pOrigin,403.64,104.03,0.00),v40,z0,tPen\WObj:=wPaper;
    MoveL Offs(pOrigin,403.85,103.60,0.00),v40,z0,tPen\WObj:=wPaper;
    MoveL Offs(pOrigin,403.99,104.11,0.00),v40,z0,tPen\WObj:=wPaper;
    MoveL Offs(pOrigin,402.34,102.45,0.00),v40,z0,tPen\WObj:=wPaper;
    MoveL Offs(pOrigin,402.58,102.65,0.00),v40,z0,tPen\WObj:=wPaper;
    MoveL Offs(pOrigin,404.28,102.65,0.00),v40,z0,tPen\WObj:=wPaper;
    MoveL Offs(pOrigin,404.58,103.21,0.00),v40,z0,tPen\WObj:=wPaper;
    MoveL Offs(pOrigin,402.93,101.56,0.00),v40,z0,tPen\WObj:=wPaper;
    MoveL Offs(pOrigin,403.42,101.59,0.00),v40,z0,tPen\WObj:=wPaper;
    MoveL Offs(pOrigin,405.12,101.59,0.00),v40,z0,tPen\WObj:=wPaper;
    MoveL Offs(pOrigin,405.78,101.41,0.00),v40,z0,tPen\WObj:=wPaper;
    MoveL Offs(pOrigin,404.12,99.76,0.00),v40,z0,tPen\WObj:=wPaper;
    MoveL Offs(pOrigin,404.49,99.78,0.00),v40,z0,tPen\WObj:=wPaper;
    MoveL Offs(pOrigin,404.27,100.20,0.00),v40,z0,tPen\WObj:=wPaper;
    MoveL Offs(pOrigin,404.49,99.78,0.00),v40,z0,tPen\WObj:=wPaper;
    MoveL Offs(pOrigin,404.70,99.48,0.00),v40,z0,tPen\WObj:=wPaper;
    MoveL Offs(pOrigin,406.40,99.48,0.00),v40,z0,tPen\WObj:=wPaper;
    MoveL Offs(pOrigin,406.82,99.47,0.00),v40,z0,tPen\WObj:=wPaper;
    MoveL Offs(pOrigin,405.02,97.67,0.00),v40,z0,tPen\WObj:=wPaper;
    MoveL Offs(pOrigin,404.44,97.59,0.00),v40,z0,tPen\WObj:=wPaper;
    MoveL Offs(pOrigin,409.85,92.18,0.00),v40,z0,tPen\WObj:=wPaper;
    MoveL Offs(pOrigin,409.49,91.69,0.00),v40,z0,tPen\WObj:=wPaper;
    MoveL Offs(pOrigin,407.39,89.59,0.00),v40,z0,tPen\WObj:=wPaper;
    MoveL Offs(pOrigin,407.89,89.98,0.00),v40,z0,tPen\WObj:=wPaper;
    MoveL Offs(pOrigin,409.38,89.98,0.00),v40,z0,tPen\WObj:=wPaper;
    MoveL Offs(pOrigin,409.79,90.49,0.00),v40,z0,tPen\WObj:=wPaper;
    MoveL Offs(pOrigin,407.84,88.54,0.00),v40,z0,tPen\WObj:=wPaper;
    MoveL Offs(pOrigin,408.10,88.92,0.00),v40,z0,tPen\WObj:=wPaper;
    MoveL Offs(pOrigin,409.80,88.92,0.00),v40,z0,tPen\WObj:=wPaper;
    MoveL Offs(pOrigin,410.08,89.29,0.00),v40,z0,tPen\WObj:=wPaper;
    MoveL Offs(pOrigin,407.98,87.19,0.00),v40,z0,tPen\WObj:=wPaper;
    MoveL Offs(pOrigin,407.62,86.95,0.00),v40,z0,tPen\WObj:=wPaper;
    MoveL Offs(pOrigin,412.58,81.99,0.00),v40,z0,tPen\WObj:=wPaper;
    MoveL Offs(pOrigin,412.01,82.26,0.00),v40,z0,tPen\WObj:=wPaper;
    MoveL Offs(pOrigin,410.06,80.31,0.00),v40,z0,tPen\WObj:=wPaper;
    MoveL Offs(pOrigin,410.44,80.47,0.00),v40,z0,tPen\WObj:=wPaper;
    MoveL Offs(pOrigin,412.14,80.47,0.00),v40,z0,tPen\WObj:=wPaper;
    MoveL Offs(pOrigin,411.85,79.80,0.00),v40,z0,tPen\WObj:=wPaper;
    MoveL Offs(pOrigin,411.85,78.52,0.00),v40,z0,tPen\WObj:=wPaper;
    MoveL Offs(pOrigin,411.29,78.36,0.00),v40,z0,tPen\WObj:=wPaper;
    MoveL Offs(pOrigin,412.99,78.36,0.00),v40,z0,tPen\WObj:=wPaper;
    MoveL Offs(pOrigin,413.35,79.12,0.00),v40,z0,tPen\WObj:=wPaper;
    MoveL Offs(pOrigin,411.40,77.16,0.00),v40,z0,tPen\WObj:=wPaper;
    MoveL Offs(pOrigin,411.71,77.30,0.00),v40,z0,tPen\WObj:=wPaper;
    MoveL Offs(pOrigin,413.41,77.30,0.00),v40,z0,tPen\WObj:=wPaper;
    MoveL Offs(pOrigin,412.91,77.46,0.00),v40,z0,tPen\WObj:=wPaper;
    MoveL Offs(pOrigin,412.91,76.19,0.00),v40,z0,tPen\WObj:=wPaper;
    MoveL Offs(pOrigin,412.35,76.25,0.00),v40,z0,tPen\WObj:=wPaper;
    MoveL Offs(pOrigin,413.84,76.25,0.00),v40,z0,tPen\WObj:=wPaper;
    MoveL Offs(pOrigin,414.09,76.87,0.00),v40,z0,tPen\WObj:=wPaper;
    MoveL Offs(pOrigin,412.14,74.92,0.00),v40,z0,tPen\WObj:=wPaper;
    MoveL Offs(pOrigin,412.78,75.19,0.00),v40,z0,tPen\WObj:=wPaper;
    MoveL Offs(pOrigin,414.26,75.19,0.00),v40,z0,tPen\WObj:=wPaper;
    MoveL Offs(pOrigin,413.97,74.70,0.00),v40,z0,tPen\WObj:=wPaper;
    MoveL Offs(pOrigin,413.97,73.21,0.00),v40,z0,tPen\WObj:=wPaper;
    MoveL Offs(pOrigin,413.41,73.08,0.00),v40,z0,tPen\WObj:=wPaper;
    MoveL Offs(pOrigin,415.11,73.08,0.00),v40,z0,tPen\WObj:=wPaper;
    MoveL Offs(pOrigin,415.43,73.73,0.00),v40,z0,tPen\WObj:=wPaper;
    MoveL Offs(pOrigin,413.33,71.63,0.00),v40,z0,tPen\WObj:=wPaper;
    MoveL Offs(pOrigin,413.84,72.02,0.00),v40,z0,tPen\WObj:=wPaper;
    MoveL Offs(pOrigin,415.54,72.02,0.00),v40,z0,tPen\WObj:=wPaper;
    MoveL Offs(pOrigin,415.73,72.53,0.00),v40,z0,tPen\WObj:=wPaper;
    MoveL Offs(pOrigin,413.62,70.43,0.00),v40,z0,tPen\WObj:=wPaper;
    MoveL Offs(pOrigin,414.05,70.97,0.00),v40,z0,tPen\WObj:=wPaper;
    MoveL Offs(pOrigin,415.75,70.97,0.00),v40,z0,tPen\WObj:=wPaper;
    MoveL Offs(pOrigin,416.02,71.34,0.00),v40,z0,tPen\WObj:=wPaper;
    MoveL Offs(pOrigin,411.66,66.98,0.00),v40,z0,tPen\WObj:=wPaper;
    MoveL Offs(pOrigin,412.14,67.05,0.00),v40,z0,tPen\WObj:=wPaper;
    MoveL Offs(pOrigin,411.29,68.11,0.00),v40,z0,tPen\WObj:=wPaper;
    MoveL Offs(pOrigin,412.14,67.05,0.00),v40,z0,tPen\WObj:=wPaper;
    MoveL Offs(pOrigin,412.35,66.74,0.00),v40,z0,tPen\WObj:=wPaper;
    MoveL Offs(pOrigin,415.96,66.74,0.00),v40,z0,tPen\WObj:=wPaper;
    MoveL Offs(pOrigin,416.46,67.29,0.00),v40,z0,tPen\WObj:=wPaper;
    MoveL Offs(pOrigin,413.30,64.14,0.00),v40,z0,tPen\WObj:=wPaper;
    MoveL Offs(pOrigin,412.79,63.86,0.00),v40,z0,tPen\WObj:=wPaper;
    MoveL Offs(pOrigin,417.44,59.20,0.00),v40,z0,tPen\WObj:=wPaper;
    MoveL Offs(pOrigin,417.03,58.91,0.00),v40,z0,tPen\WObj:=wPaper;
    MoveL Offs(pOrigin,414.33,56.20,0.00),v40,z0,tPen\WObj:=wPaper;
    MoveL Offs(pOrigin,414.01,56.67,0.00),v40,z0,tPen\WObj:=wPaper;
    MoveL Offs(pOrigin,417.31,53.36,0.00),v40,z0,tPen\WObj:=wPaper;
    MoveL Offs(pOrigin,416.72,52.46,0.00),v40,z0,tPen\WObj:=wPaper;
    MoveL Offs(pOrigin,414.01,55.17,0.00),v40,z0,tPen\WObj:=wPaper;
    MoveL Offs(pOrigin,414.90,55.13,0.00),v40,z0,tPen\WObj:=wPaper;
    MoveL Offs(pOrigin,416.39,55.13,0.00),v40,z0,tPen\WObj:=wPaper;
    MoveL Offs(pOrigin,417.02,55.91,0.00),v40,z0,tPen\WObj:=wPaper;
    MoveL Offs(pOrigin,414.02,52.91,0.00),v40,z0,tPen\WObj:=wPaper;
    MoveL Offs(pOrigin,413.57,52.62,0.00),v40,z0,tPen\WObj:=wPaper;
    MoveL Offs(pOrigin,416.27,49.92,0.00),v40,z0,tPen\WObj:=wPaper;
    MoveL Offs(pOrigin,415.96,50.36,0.00),v40,z0,tPen\WObj:=wPaper;
    MoveL Offs(pOrigin,402.88,37.29,0.00),v40,z0,tPen\WObj:=wPaper;
    MoveL Offs(pOrigin,402.68,36.63,0.00),v40,z0,tPen\WObj:=wPaper;
    MoveL Offs(pOrigin,400.28,39.03,0.00),v40,z0,tPen\WObj:=wPaper;
    MoveL Offs(pOrigin,399.59,38.48,0.00),v40,z0,tPen\WObj:=wPaper;
    MoveL Offs(pOrigin,396.74,35.63,0.00),v40,z0,tPen\WObj:=wPaper;
    MoveL Offs(pOrigin,396.85,35.00,0.00),v40,z0,tPen\WObj:=wPaper;
    MoveL Offs(pOrigin,394.44,37.40,0.00),v40,z0,tPen\WObj:=wPaper;
    MoveL Offs(pOrigin,395.54,37.42,0.00),v40,z0,tPen\WObj:=wPaper;
    MoveL Offs(pOrigin,392.84,34.71,0.00),v40,z0,tPen\WObj:=wPaper;
    MoveL Offs(pOrigin,392.80,35.06,0.00),v40,z0,tPen\WObj:=wPaper;
    MoveL Offs(pOrigin,387.49,35.06,0.00),v40,z0,tPen\WObj:=wPaper;
    MoveL Offs(pOrigin,388.05,35.90,0.00),v40,z0,tPen\WObj:=wPaper;
    MoveL Offs(pOrigin,385.50,33.34,0.00),v40,z0,tPen\WObj:=wPaper;
    MoveL Offs(pOrigin,385.62,32.79,0.00),v40,z0,tPen\WObj:=wPaper;
    MoveL Offs(pOrigin,383.06,35.34,0.00),v40,z0,tPen\WObj:=wPaper;
    MoveL Offs(pOrigin,382.65,34.98,0.00),v40,z0,tPen\WObj:=wPaper;
    MoveL Offs(pOrigin,380.10,32.43,0.00),v40,z0,tPen\WObj:=wPaper;
    MoveL Offs(pOrigin,380.48,32.95,0.00),v40,z0,tPen\WObj:=wPaper;
  ENDPROC

  PROC DrawPart64()
    MoveL Offs(pOrigin,372.61,32.95,0.00),v40,z0,tPen\WObj:=wPaper;
    MoveL Offs(pOrigin,372.61,33.90,0.00),v40,z0,tPen\WObj:=wPaper;
    MoveL Offs(pOrigin,370.21,31.50,0.00),v40,z0,tPen\WObj:=wPaper;
    MoveL Offs(pOrigin,369.74,30.74,0.00),v40,z0,tPen\WObj:=wPaper;
    MoveL Offs(pOrigin,365.99,34.49,0.00),v40,z0,tPen\WObj:=wPaper;
    MoveL Offs(pOrigin,367.04,34.94,0.00),v40,z0,tPen\WObj:=wPaper;
    MoveL Offs(pOrigin,371.09,30.88,0.00),v40,z0,tPen\WObj:=wPaper;
    MoveL Offs(pOrigin,371.56,31.35,0.00),v40,z0,tPen\WObj:=wPaper;
    MoveL Offs(pOrigin,373.96,33.76,0.00),v40,fine,tPen\WObj:=wPaper;
    MoveL Offs(pOrigin,373.96,33.76,6.00),v60,z5,tPen\WObj:=wPaper;
    MoveL Offs(pOrigin,375.00,31.81,6.00),vTravel,z5,tPen\WObj:=wPaper;
    MoveL Offs(pOrigin,375.00,31.81,0.00),v60,z0,tPen\WObj:=wPaper;
    MoveL Offs(pOrigin,377.41,34.22,0.00),v40,z0,tPen\WObj:=wPaper;
    MoveL Offs(pOrigin,377.67,34.76,0.00),v40,z0,tPen\WObj:=wPaper;
    MoveL Offs(pOrigin,380.53,31.90,0.00),v40,fine,tPen\WObj:=wPaper;
    MoveL Offs(pOrigin,380.53,31.90,6.00),v60,z5,tPen\WObj:=wPaper;
    MoveL Offs(pOrigin,381.87,32.05,6.00),vTravel,z5,tPen\WObj:=wPaper;
    MoveL Offs(pOrigin,381.87,32.05,0.00),v60,z0,tPen\WObj:=wPaper;
    MoveL Offs(pOrigin,379.02,34.90,0.00),v40,z0,tPen\WObj:=wPaper;
    MoveL Offs(pOrigin,379.06,34.37,0.00),v40,z0,tPen\WObj:=wPaper;
    MoveL Offs(pOrigin,376.65,31.97,0.00),v40,z0,tPen\WObj:=wPaper;
    MoveL Offs(pOrigin,376.48,31.47,0.00),v40,z0,tPen\WObj:=wPaper;
    MoveL Offs(pOrigin,371.53,36.42,0.00),v40,z0,tPen\WObj:=wPaper;
    MoveL Offs(pOrigin,372.17,36.45,0.00),v40,z0,tPen\WObj:=wPaper;
    MoveL Offs(pOrigin,366.76,31.04,0.00),v40,z0,tPen\WObj:=wPaper;
    MoveL Offs(pOrigin,367.05,30.45,0.00),v40,z0,tPen\WObj:=wPaper;
    MoveL Offs(pOrigin,363.74,33.75,0.00),v40,z0,tPen\WObj:=wPaper;
    MoveL Offs(pOrigin,364.33,32.95,0.00),v40,z0,tPen\WObj:=wPaper;
    MoveL Offs(pOrigin,368.79,32.95,0.00),v40,z0,tPen\WObj:=wPaper;
    MoveL Offs(pOrigin,369.21,34.01,0.00),v40,z0,tPen\WObj:=wPaper;
    MoveL Offs(pOrigin,367.94,34.01,0.00),v40,z0,tPen\WObj:=wPaper;
    MoveL Offs(pOrigin,367.67,34.94,0.00),v40,z0,tPen\WObj:=wPaper;
    MoveL Offs(pOrigin,362.87,30.13,0.00),v40,z0,tPen\WObj:=wPaper;
    MoveL Offs(pOrigin,363.31,29.71,0.00),v40,z0,tPen\WObj:=wPaper;
    MoveL Offs(pOrigin,360.75,32.26,0.00),v40,z0,tPen\WObj:=wPaper;
    MoveL Offs(pOrigin,360.18,31.92,0.00),v40,z0,tPen\WObj:=wPaper;
    MoveL Offs(pOrigin,355.82,27.56,0.00),v40,z0,tPen\WObj:=wPaper;
    MoveL Offs(pOrigin,355.40,27.67,0.00),v40,z0,tPen\WObj:=wPaper;
    MoveL Offs(pOrigin,353.06,27.67,0.00),v40,z0,tPen\WObj:=wPaper;
    MoveL Offs(pOrigin,352.52,28.54,0.00),v40,z0,tPen\WObj:=wPaper;
    MoveL Offs(pOrigin,354.78,26.29,0.00),v40,z0,tPen\WObj:=wPaper;
    MoveL Offs(pOrigin,355.83,26.74,0.00),v40,z0,tPen\WObj:=wPaper;
    MoveL Offs(pOrigin,353.57,28.99,0.00),v40,z0,tPen\WObj:=wPaper;
    MoveL Offs(pOrigin,354.47,29.59,0.00),v40,z0,tPen\WObj:=wPaper;
    MoveL Offs(pOrigin,356.87,27.18,0.00),v40,fine,tPen\WObj:=wPaper;
    MoveL Offs(pOrigin,356.87,27.18,6.00),v60,z5,tPen\WObj:=wPaper;
    MoveL Offs(pOrigin,353.73,25.84,6.00),vTravel,z5,tPen\WObj:=wPaper;
    MoveL Offs(pOrigin,353.73,25.84,0.00),v60,z0,tPen\WObj:=wPaper;
    MoveL Offs(pOrigin,351.48,28.10,0.00),v40,z0,tPen\WObj:=wPaper;
    MoveL Offs(pOrigin,351.62,27.85,0.00),v40,z0,tPen\WObj:=wPaper;
    MoveL Offs(pOrigin,348.17,24.39,0.00),v40,z0,tPen\WObj:=wPaper;
    MoveL Offs(pOrigin,348.35,23.76,0.00),v40,z0,tPen\WObj:=wPaper;
    MoveL Offs(pOrigin,340.83,31.28,0.00),v40,z0,tPen\WObj:=wPaper;
    MoveL Offs(pOrigin,341.15,30.81,0.00),v40,z0,tPen\WObj:=wPaper;
    MoveL Offs(pOrigin,335.74,25.40,0.00),v40,z0,tPen\WObj:=wPaper;
    MoveL Offs(pOrigin,335.31,24.85,0.00),v40,z0,tPen\WObj:=wPaper;
    MoveL Offs(pOrigin,331.25,28.91,0.00),v40,z0,tPen\WObj:=wPaper;
    MoveL Offs(pOrigin,331.25,28.38,0.00),v40,z0,tPen\WObj:=wPaper;
    MoveL Offs(pOrigin,328.85,25.98,0.00),v40,z0,tPen\WObj:=wPaper;
    MoveL Offs(pOrigin,328.87,25.32,0.00),v40,z0,tPen\WObj:=wPaper;
    MoveL Offs(pOrigin,326.16,28.03,0.00),v40,fine,tPen\WObj:=wPaper;
    MoveL Offs(pOrigin,326.16,28.03,6.00),v60,z5,tPen\WObj:=wPaper;
    MoveL Offs(pOrigin,324.96,27.73,6.00),vTravel,z5,tPen\WObj:=wPaper;
    MoveL Offs(pOrigin,324.96,27.73,0.00),v60,z0,tPen\WObj:=wPaper;
    MoveL Offs(pOrigin,327.52,25.18,0.00),v40,z0,tPen\WObj:=wPaper;
    MoveL Offs(pOrigin,327.05,25.67,0.00),v40,z0,tPen\WObj:=wPaper;
    MoveL Offs(pOrigin,329.45,28.08,0.00),v40,z0,tPen\WObj:=wPaper;
    MoveL Offs(pOrigin,328.86,28.32,0.00),v40,z0,tPen\WObj:=wPaper;
    MoveL Offs(pOrigin,331.41,25.76,0.00),v40,z0,tPen\WObj:=wPaper;
    MoveL Offs(pOrigin,332.30,26.44,0.00),v40,z0,tPen\WObj:=wPaper;
    MoveL Offs(pOrigin,335.00,29.14,0.00),v40,z0,tPen\WObj:=wPaper;
    MoveL Offs(pOrigin,334.99,29.65,0.00),v40,z0,tPen\WObj:=wPaper;
    MoveL Offs(pOrigin,341.46,23.18,0.00),v40,z0,tPen\WObj:=wPaper;
    MoveL Offs(pOrigin,341.57,23.77,0.00),v40,z0,tPen\WObj:=wPaper;
    MoveL Offs(pOrigin,350.74,32.94,0.00),v40,z0,tPen\WObj:=wPaper;
    MoveL Offs(pOrigin,351.46,32.59,0.00),v40,z0,tPen\WObj:=wPaper;
    MoveL Offs(pOrigin,346.35,37.70,0.00),v40,z0,tPen\WObj:=wPaper;
    MoveL Offs(pOrigin,347.01,38.17,0.00),v40,z0,tPen\WObj:=wPaper;
    MoveL Offs(pOrigin,350.47,41.63,0.00),v40,z0,tPen\WObj:=wPaper;
    MoveL Offs(pOrigin,350.68,42.33,0.00),v40,z0,tPen\WObj:=wPaper;
    MoveL Offs(pOrigin,341.82,51.20,0.00),v40,z0,tPen\WObj:=wPaper;
    MoveL Offs(pOrigin,342.56,51.64,0.00),v40,z0,tPen\WObj:=wPaper;
    MoveL Offs(pOrigin,343.91,52.99,0.00),v40,z0,tPen\WObj:=wPaper;
    MoveL Offs(pOrigin,343.50,53.02,0.00),v40,z0,tPen\WObj:=wPaper;
    MoveL Offs(pOrigin,342.22,53.02,0.00),v40,z0,tPen\WObj:=wPaper;
    MoveL Offs(pOrigin,341.96,52.53,0.00),v40,z0,tPen\WObj:=wPaper;
    MoveL Offs(pOrigin,343.32,53.89,0.00),v40,z0,tPen\WObj:=wPaper;
    MoveL Offs(pOrigin,342.65,54.07,0.00),v40,z0,tPen\WObj:=wPaper;
    MoveL Offs(pOrigin,341.38,54.07,0.00),v40,z0,tPen\WObj:=wPaper;
    MoveL Offs(pOrigin,340.62,54.18,0.00),v40,z0,tPen\WObj:=wPaper;
    MoveL Offs(pOrigin,342.12,55.68,0.00),v40,z0,tPen\WObj:=wPaper;
    MoveL Offs(pOrigin,341.80,55.13,0.00),v40,z0,tPen\WObj:=wPaper;
    MoveL Offs(pOrigin,340.52,55.13,0.00),v40,z0,tPen\WObj:=wPaper;
    MoveL Offs(pOrigin,340.52,54.72,0.00),v40,z0,tPen\WObj:=wPaper;
    MoveL Offs(pOrigin,339.89,55.36,0.00),v40,z0,tPen\WObj:=wPaper;
    MoveL Offs(pOrigin,340.52,54.72,0.00),v40,z0,tPen\WObj:=wPaper;
    MoveL Offs(pOrigin,339.87,54.92,0.00),v40,z0,tPen\WObj:=wPaper;
    MoveL Offs(pOrigin,341.53,56.58,0.00),v40,z0,tPen\WObj:=wPaper;
    MoveL Offs(pOrigin,340.95,56.18,0.00),v40,z0,tPen\WObj:=wPaper;
    MoveL Offs(pOrigin,339.67,56.18,0.00),v40,z0,tPen\WObj:=wPaper;
    MoveL Offs(pOrigin,339.67,55.79,0.00),v40,z0,tPen\WObj:=wPaper;
    MoveL Offs(pOrigin,339.25,56.21,0.00),v40,z0,tPen\WObj:=wPaper;
    MoveL Offs(pOrigin,339.67,55.79,0.00),v40,z0,tPen\WObj:=wPaper;
    MoveL Offs(pOrigin,339.28,55.82,0.00),v40,z0,tPen\WObj:=wPaper;
    MoveL Offs(pOrigin,340.63,57.17,0.00),v40,z0,tPen\WObj:=wPaper;
    MoveL Offs(pOrigin,340.10,57.24,0.00),v40,z0,tPen\WObj:=wPaper;
    MoveL Offs(pOrigin,338.61,57.24,0.00),v40,z0,tPen\WObj:=wPaper;
    MoveL Offs(pOrigin,338.53,56.57,0.00),v40,z0,tPen\WObj:=wPaper;
    MoveL Offs(pOrigin,340.03,58.07,0.00),v40,z0,tPen\WObj:=wPaper;
    MoveL Offs(pOrigin,340.03,57.63,0.00),v40,z0,tPen\WObj:=wPaper;
    MoveL Offs(pOrigin,337.98,59.61,0.00),v40,z0,tPen\WObj:=wPaper;
    MoveL Offs(pOrigin,340.03,57.63,0.00),v40,z0,tPen\WObj:=wPaper;
    MoveL Offs(pOrigin,341.20,57.79,0.00),v40,z0,tPen\WObj:=wPaper;
    MoveL Offs(pOrigin,338.04,60.94,0.00),v40,z0,tPen\WObj:=wPaper;
    MoveL Offs(pOrigin,337.64,60.16,0.00),v40,z0,tPen\WObj:=wPaper;
    MoveL Offs(pOrigin,336.29,58.81,0.00),v40,z0,tPen\WObj:=wPaper;
    MoveL Offs(pOrigin,336.49,59.35,0.00),v40,z0,tPen\WObj:=wPaper;
    MoveL Offs(pOrigin,337.98,59.35,0.00),v40,z0,tPen\WObj:=wPaper;
    MoveL Offs(pOrigin,338.54,59.56,0.00),v40,z0,tPen\WObj:=wPaper;
    MoveL Offs(pOrigin,337.04,58.06,0.00),v40,z0,tPen\WObj:=wPaper;
  ENDPROC

  PROC DrawPart65()
    MoveL Offs(pOrigin,337.34,58.12,0.00),v40,z0,tPen\WObj:=wPaper;
    MoveL Offs(pOrigin,335.85,59.61,0.00),v40,z0,tPen\WObj:=wPaper;
    MoveL Offs(pOrigin,337.34,58.12,0.00),v40,z0,tPen\WObj:=wPaper;
    MoveL Offs(pOrigin,337.55,58.30,0.00),v40,z0,tPen\WObj:=wPaper;
    MoveL Offs(pOrigin,339.04,58.30,0.00),v40,z0,tPen\WObj:=wPaper;
    MoveL Offs(pOrigin,339.44,58.97,0.00),v40,z0,tPen\WObj:=wPaper;
    MoveL Offs(pOrigin,337.78,57.32,0.00),v40,fine,tPen\WObj:=wPaper;
    MoveL Offs(pOrigin,337.78,57.32,6.00),v60,z5,tPen\WObj:=wPaper;
    MoveL Offs(pOrigin,339.04,56.42,6.00),vTravel,z5,tPen\WObj:=wPaper;
    MoveL Offs(pOrigin,339.04,56.42,0.00),v60,z0,tPen\WObj:=wPaper;
    MoveL Offs(pOrigin,337.55,57.91,0.00),v40,z0,tPen\WObj:=wPaper;
    MoveL Offs(pOrigin,339.04,56.42,0.00),v40,fine,tPen\WObj:=wPaper;
    MoveL Offs(pOrigin,339.04,56.42,6.00),v60,z5,tPen\WObj:=wPaper;
    MoveL Offs(pOrigin,337.17,54.36,6.00),vTravel,z5,tPen\WObj:=wPaper;
    MoveL Offs(pOrigin,337.17,54.36,0.00),v60,z0,tPen\WObj:=wPaper;
    MoveL Offs(pOrigin,334.01,57.51,0.00),v40,fine,tPen\WObj:=wPaper;
    MoveL Offs(pOrigin,334.01,57.51,6.00),v60,z5,tPen\WObj:=wPaper;
    MoveL Offs(pOrigin,334.01,59.01,6.00),vTravel,z5,tPen\WObj:=wPaper;
    MoveL Offs(pOrigin,334.01,59.01,0.00),v60,z0,tPen\WObj:=wPaper;
    MoveL Offs(pOrigin,324.09,68.93,0.00),v40,z0,tPen\WObj:=wPaper;
    MoveL Offs(pOrigin,323.59,68.51,0.00),v40,z0,tPen\WObj:=wPaper;
    MoveL Offs(pOrigin,321.93,66.85,0.00),v40,z0,tPen\WObj:=wPaper;
    MoveL Offs(pOrigin,322.98,66.41,0.00),v40,z0,tPen\WObj:=wPaper;
    MoveL Offs(pOrigin,324.78,68.21,0.00),v40,z0,tPen\WObj:=wPaper;
    MoveL Offs(pOrigin,323.74,67.80,0.00),v40,z0,tPen\WObj:=wPaper;
    MoveL Offs(pOrigin,310.99,67.80,0.00),v40,z0,tPen\WObj:=wPaper;
    MoveL Offs(pOrigin,311.53,67.90,0.00),v40,z0,tPen\WObj:=wPaper;
    MoveL Offs(pOrigin,311.53,66.84,0.00),v40,z0,tPen\WObj:=wPaper;
    MoveL Offs(pOrigin,312.59,66.84,0.00),v40,z0,tPen\WObj:=wPaper;
    MoveL Offs(pOrigin,312.59,68.54,0.00),v40,z0,tPen\WObj:=wPaper;
    MoveL Offs(pOrigin,312.69,68.86,0.00),v40,z0,tPen\WObj:=wPaper;
    MoveL Offs(pOrigin,316.94,68.86,0.00),v40,z0,tPen\WObj:=wPaper;
    MoveL Offs(pOrigin,316.30,68.75,0.00),v40,z0,tPen\WObj:=wPaper;
    MoveL Offs(pOrigin,314.17,68.11,0.00),v40,z0,tPen\WObj:=wPaper;
    MoveL Offs(pOrigin,313.65,68.96,0.00),v40,z0,tPen\WObj:=wPaper;
    MoveL Offs(pOrigin,313.65,67.05,0.00),v40,fine,tPen\WObj:=wPaper;
    MoveL Offs(pOrigin,313.65,67.05,6.00),v60,z5,tPen\WObj:=wPaper;
    MoveL Offs(pOrigin,312.48,69.18,6.00),vTravel,z5,tPen\WObj:=wPaper;
    MoveL Offs(pOrigin,312.48,69.18,0.00),v60,z0,tPen\WObj:=wPaper;
    MoveL Offs(pOrigin,312.90,69.39,0.00),v40,z0,tPen\WObj:=wPaper;
    MoveL Offs(pOrigin,312.48,69.18,0.00),v40,z0,tPen\WObj:=wPaper;
    MoveL Offs(pOrigin,312.55,70.01,0.00),v40,z0,tPen\WObj:=wPaper;
    MoveL Offs(pOrigin,316.46,66.10,0.00),v40,fine,tPen\WObj:=wPaper;
    MoveL Offs(pOrigin,316.46,66.10,6.00),v60,z5,tPen\WObj:=wPaper;
    MoveL Offs(pOrigin,319.09,66.99,6.00),vTravel,z5,tPen\WObj:=wPaper;
    MoveL Offs(pOrigin,319.09,66.99,0.00),v60,z0,tPen\WObj:=wPaper;
    MoveL Offs(pOrigin,321.19,69.10,0.00),v40,fine,tPen\WObj:=wPaper;
    MoveL Offs(pOrigin,321.19,69.10,6.00),v60,z5,tPen\WObj:=wPaper;
    MoveL Offs(pOrigin,322.39,68.80,6.00),vTravel,z5,tPen\WObj:=wPaper;
    MoveL Offs(pOrigin,322.39,68.80,0.00),v60,z0,tPen\WObj:=wPaper;
    MoveL Offs(pOrigin,320.59,67.00,0.00),v40,z0,tPen\WObj:=wPaper;
    MoveL Offs(pOrigin,320.80,66.24,0.00),v40,z0,tPen\WObj:=wPaper;
    MoveL Offs(pOrigin,315.69,71.35,0.00),v40,z0,tPen\WObj:=wPaper;
    MoveL Offs(pOrigin,315.35,70.73,0.00),v40,z0,tPen\WObj:=wPaper;
    MoveL Offs(pOrigin,309.94,65.32,0.00),v40,z0,tPen\WObj:=wPaper;
    MoveL Offs(pOrigin,309.19,64.57,0.00),v40,z0,tPen\WObj:=wPaper;
    MoveL Offs(pOrigin,304.08,59.46,0.00),v40,z0,tPen\WObj:=wPaper;
    MoveL Offs(pOrigin,304.50,58.65,0.00),v40,z0,tPen\WObj:=wPaper;
    MoveL Offs(pOrigin,298.79,64.36,0.00),v40,z0,tPen\WObj:=wPaper;
    MoveL Offs(pOrigin,299.73,64.07,0.00),v40,z0,tPen\WObj:=wPaper;
    MoveL Offs(pOrigin,300.36,64.50,0.00),v40,z0,tPen\WObj:=wPaper;
    MoveL Offs(pOrigin,299.73,64.07,0.00),v40,z0,tPen\WObj:=wPaper;
    MoveL Offs(pOrigin,299.68,64.96,0.00),v40,z0,tPen\WObj:=wPaper;
    MoveL Offs(pOrigin,305.99,58.65,0.00),v40,z0,tPen\WObj:=wPaper;
    MoveL Offs(pOrigin,305.43,59.31,0.00),v40,z0,tPen\WObj:=wPaper;
    MoveL Offs(pOrigin,310.39,64.27,0.00),v40,fine,tPen\WObj:=wPaper;
    MoveL Offs(pOrigin,310.39,64.27,6.00),v60,z5,tPen\WObj:=wPaper;
    MoveL Offs(pOrigin,308.65,65.69,6.00),vTravel,z5,tPen\WObj:=wPaper;
    MoveL Offs(pOrigin,308.65,65.69,0.00),v60,z0,tPen\WObj:=wPaper;
    MoveL Offs(pOrigin,304.19,65.69,0.00),v40,z0,tPen\WObj:=wPaper;
    MoveL Offs(pOrigin,303.36,66.20,0.00),v40,z0,tPen\WObj:=wPaper;
    MoveL Offs(pOrigin,297.95,60.79,0.00),v40,z0,tPen\WObj:=wPaper;
    MoveL Offs(pOrigin,298.86,61.52,0.00),v40,z0,tPen\WObj:=wPaper;
    MoveL Offs(pOrigin,298.86,62.59,0.00),v40,fine,tPen\WObj:=wPaper;
    MoveL Offs(pOrigin,298.86,62.59,6.00),v60,z5,tPen\WObj:=wPaper;
    MoveL Offs(pOrigin,300.36,62.16,6.00),vTravel,z5,tPen\WObj:=wPaper;
    MoveL Offs(pOrigin,300.36,62.16,0.00),v60,z0,tPen\WObj:=wPaper;
    MoveL Offs(pOrigin,302.91,64.00,0.00),v40,z0,tPen\WObj:=wPaper;
    MoveL Offs(pOrigin,310.35,65.99,0.00),v40,z0,tPen\WObj:=wPaper;
    MoveL Offs(pOrigin,318.21,67.26,0.00),v40,z0,tPen\WObj:=wPaper;
    MoveL Offs(pOrigin,321.40,67.26,0.00),v40,z0,tPen\WObj:=wPaper;
    MoveL Offs(pOrigin,325.01,66.27,0.00),v40,z0,tPen\WObj:=wPaper;
    MoveL Offs(pOrigin,330.54,63.72,0.00),v40,z0,tPen\WObj:=wPaper;
    MoveL Offs(pOrigin,336.06,59.61,0.00),v40,z0,tPen\WObj:=wPaper;
    MoveL Offs(pOrigin,340.74,54.72,0.00),v40,z0,tPen\WObj:=wPaper;
    MoveL Offs(pOrigin,344.63,49.20,0.00),v40,z0,tPen\WObj:=wPaper;
    MoveL Offs(pOrigin,346.76,45.59,0.00),v40,z0,tPen\WObj:=wPaper;
    MoveL Offs(pOrigin,347.75,43.04,0.00),v40,z0,tPen\WObj:=wPaper;
    MoveL Offs(pOrigin,347.75,39.85,0.00),v40,z0,tPen\WObj:=wPaper;
    MoveL Offs(pOrigin,346.12,34.54,0.00),v40,z0,tPen\WObj:=wPaper;
    MoveL Offs(pOrigin,344.14,31.99,0.00),v40,z0,tPen\WObj:=wPaper;
    MoveL Offs(pOrigin,341.16,30.43,0.00),v40,z0,tPen\WObj:=wPaper;
    MoveL Offs(pOrigin,336.27,29.01,0.00),v40,z0,tPen\WObj:=wPaper;
    MoveL Offs(pOrigin,322.04,26.46,0.00),v40,z0,tPen\WObj:=wPaper;
    MoveL Offs(pOrigin,319.27,26.25,0.00),v40,z0,tPen\WObj:=wPaper;
    MoveL Offs(pOrigin,318.85,26.67,0.00),v40,z0,tPen\WObj:=wPaper;
    MoveL Offs(pOrigin,318.85,26.67,0.00),v40,z0,tPen\WObj:=wPaper;
    MoveL Offs(pOrigin,320.34,27.52,0.00),v40,z0,tPen\WObj:=wPaper;
    MoveL Offs(pOrigin,321.40,28.59,0.00),v40,z0,tPen\WObj:=wPaper;
    MoveL Offs(pOrigin,323.17,31.77,0.00),v40,z0,tPen\WObj:=wPaper;
    MoveL Offs(pOrigin,324.80,38.79,0.00),v40,z0,tPen\WObj:=wPaper;
    MoveL Offs(pOrigin,324.80,44.10,0.00),v40,z0,tPen\WObj:=wPaper;
    MoveL Offs(pOrigin,323.52,50.47,0.00),v40,z0,tPen\WObj:=wPaper;
    MoveL Offs(pOrigin,321.90,55.15,0.00),v40,z0,tPen\WObj:=wPaper;
    MoveL Offs(pOrigin,320.05,58.34,0.00),v40,z0,tPen\WObj:=wPaper;
    MoveL Offs(pOrigin,318.00,60.67,0.00),v40,z0,tPen\WObj:=wPaper;
    MoveL Offs(pOrigin,317.58,60.41,0.00),v40,z0,tPen\WObj:=wPaper;
    MoveL Offs(pOrigin,301.00,60.41,0.00),v40,z0,tPen\WObj:=wPaper;
    MoveL Offs(pOrigin,300.49,60.35,0.00),v40,z0,tPen\WObj:=wPaper;
    MoveL Offs(pOrigin,307.55,67.41,0.00),v40,z0,tPen\WObj:=wPaper;
    MoveL Offs(pOrigin,307.47,67.63,0.00),v40,z0,tPen\WObj:=wPaper;
    MoveL Offs(pOrigin,324.14,50.95,0.00),v40,z0,tPen\WObj:=wPaper;
    MoveL Offs(pOrigin,323.68,50.68,0.00),v40,z0,tPen\WObj:=wPaper;
    MoveL Offs(pOrigin,321.73,48.73,0.00),v40,z0,tPen\WObj:=wPaper;
    MoveL Offs(pOrigin,320.86,48.26,0.00),v40,z0,tPen\WObj:=wPaper;
    MoveL Offs(pOrigin,325.67,43.46,0.00),v40,z0,tPen\WObj:=wPaper;
    MoveL Offs(pOrigin,324.86,42.89,0.00),v40,z0,tPen\WObj:=wPaper;
    MoveL Offs(pOrigin,322.75,40.79,0.00),v40,z0,tPen\WObj:=wPaper;
    MoveL Offs(pOrigin,322.89,40.28,0.00),v40,z0,tPen\WObj:=wPaper;
    MoveL Offs(pOrigin,322.46,36.66,0.00),v40,z0,tPen\WObj:=wPaper;
  ENDPROC

  PROC DrawPart66()
    MoveL Offs(pOrigin,321.75,36.03,0.00),v40,z0,tPen\WObj:=wPaper;
    MoveL Offs(pOrigin,321.26,34.75,0.00),v40,z0,tPen\WObj:=wPaper;
    MoveL Offs(pOrigin,321.40,34.33,0.00),v40,z0,tPen\WObj:=wPaper;
    MoveL Offs(pOrigin,321.40,34.33,0.00),v40,z0,tPen\WObj:=wPaper;
    MoveL Offs(pOrigin,320.34,32.62,0.00),v40,z0,tPen\WObj:=wPaper;
    MoveL Offs(pOrigin,319.27,31.92,0.00),v40,z0,tPen\WObj:=wPaper;
    MoveL Offs(pOrigin,313.96,29.72,0.00),v40,z0,tPen\WObj:=wPaper;
    MoveL Offs(pOrigin,313.89,30.50,0.00),v40,z0,tPen\WObj:=wPaper;
    MoveL Offs(pOrigin,315.95,34.11,0.00),v40,z0,tPen\WObj:=wPaper;
    MoveL Offs(pOrigin,315.88,34.96,0.00),v40,fine,tPen\WObj:=wPaper;
    MoveL Offs(pOrigin,315.88,34.96,6.00),v60,z5,tPen\WObj:=wPaper;
    MoveL Offs(pOrigin,314.61,32.11,6.00),vTravel,z5,tPen\WObj:=wPaper;
    MoveL Offs(pOrigin,314.61,32.11,0.00),v60,z0,tPen\WObj:=wPaper;
    MoveL Offs(pOrigin,322.58,24.14,0.00),v40,z0,tPen\WObj:=wPaper;
    MoveL Offs(pOrigin,321.65,24.76,0.00),v40,z0,tPen\WObj:=wPaper;
    MoveL Offs(pOrigin,324.06,27.16,0.00),v40,z0,tPen\WObj:=wPaper;
    MoveL Offs(pOrigin,323.62,27.58,0.00),v40,z0,tPen\WObj:=wPaper;
    MoveL Offs(pOrigin,326.32,24.88,0.00),v40,z0,tPen\WObj:=wPaper;
    MoveL Offs(pOrigin,325.25,25.37,0.00),v40,z0,tPen\WObj:=wPaper;
    MoveL Offs(pOrigin,327.51,27.62,0.00),v40,z0,tPen\WObj:=wPaper;
    MoveL Offs(pOrigin,327.51,28.17,0.00),v40,z0,tPen\WObj:=wPaper;
    MoveL Offs(pOrigin,330.06,25.62,0.00),v40,fine,tPen\WObj:=wPaper;
    MoveL Offs(pOrigin,330.06,25.62,6.00),v60,z5,tPen\WObj:=wPaper;
    MoveL Offs(pOrigin,330.75,27.67,6.00),vTravel,z5,tPen\WObj:=wPaper;
    MoveL Offs(pOrigin,330.75,27.67,0.00),v60,z0,tPen\WObj:=wPaper;
    MoveL Offs(pOrigin,341.80,27.67,0.00),v40,fine,tPen\WObj:=wPaper;
    MoveL Offs(pOrigin,341.80,27.67,6.00),v60,z5,tPen\WObj:=wPaper;
    MoveL Offs(pOrigin,343.29,28.16,6.00),vTravel,z5,tPen\WObj:=wPaper;
    MoveL Offs(pOrigin,343.29,28.16,0.00),v60,z0,tPen\WObj:=wPaper;
    MoveL Offs(pOrigin,345.20,29.86,0.00),v40,z0,tPen\WObj:=wPaper;
    MoveL Offs(pOrigin,343.29,28.16,0.00),v40,z0,tPen\WObj:=wPaper;
    MoveL Offs(pOrigin,343.71,28.73,0.00),v40,z0,tPen\WObj:=wPaper;
    MoveL Offs(pOrigin,335.85,28.73,0.00),v40,z0,tPen\WObj:=wPaper;
    MoveL Offs(pOrigin,335.82,28.16,0.00),v40,z0,tPen\WObj:=wPaper;
    MoveL Offs(pOrigin,335.82,26.46,0.00),v40,z0,tPen\WObj:=wPaper;
    MoveL Offs(pOrigin,336.49,25.56,0.00),v40,z0,tPen\WObj:=wPaper;
    MoveL Offs(pOrigin,339.67,25.56,0.00),v40,fine,tPen\WObj:=wPaper;
    MoveL Offs(pOrigin,339.67,25.56,6.00),v60,z5,tPen\WObj:=wPaper;
    MoveL Offs(pOrigin,337.98,24.66,6.00),vTravel,z5,tPen\WObj:=wPaper;
    MoveL Offs(pOrigin,337.98,24.66,0.00),v60,z0,tPen\WObj:=wPaper;
    MoveL Offs(pOrigin,351.06,37.73,0.00),v40,z0,tPen\WObj:=wPaper;
    MoveL Offs(pOrigin,350.72,37.18,0.00),v40,z0,tPen\WObj:=wPaper;
    MoveL Offs(pOrigin,349.66,37.18,0.00),v40,z0,tPen\WObj:=wPaper;
    MoveL Offs(pOrigin,348.60,37.18,0.00),v40,z0,tPen\WObj:=wPaper;
    MoveL Offs(pOrigin,347.54,37.18,0.00),v40,z0,tPen\WObj:=wPaper;
    MoveL Offs(pOrigin,347.75,38.23,0.00),v40,z0,tPen\WObj:=wPaper;
    MoveL Offs(pOrigin,350.51,38.23,0.00),v40,z0,tPen\WObj:=wPaper;
    MoveL Offs(pOrigin,350.51,39.29,0.00),v40,z0,tPen\WObj:=wPaper;
    MoveL Offs(pOrigin,347.96,39.29,0.00),v40,z0,tPen\WObj:=wPaper;
    MoveL Offs(pOrigin,347.96,40.34,0.00),v40,z0,tPen\WObj:=wPaper;
    MoveL Offs(pOrigin,350.30,40.34,0.00),v40,z0,tPen\WObj:=wPaper;
    MoveL Offs(pOrigin,350.76,40.43,0.00),v40,z0,tPen\WObj:=wPaper;
    MoveL Offs(pOrigin,346.11,35.77,0.00),v40,z0,tPen\WObj:=wPaper;
    MoveL Offs(pOrigin,345.61,35.46,0.00),v40,z0,tPen\WObj:=wPaper;
    MoveL Offs(pOrigin,350.42,30.65,0.00),v40,z0,tPen\WObj:=wPaper;
    MoveL Offs(pOrigin,350.94,30.29,0.00),v40,z0,tPen\WObj:=wPaper;
    MoveL Offs(pOrigin,352.92,33.69,0.00),v40,z0,tPen\WObj:=wPaper;
    MoveL Offs(pOrigin,354.12,36.88,0.00),v40,z0,tPen\WObj:=wPaper;
    MoveL Offs(pOrigin,354.55,38.79,0.00),v40,z0,tPen\WObj:=wPaper;
    MoveL Offs(pOrigin,354.34,43.25,0.00),v40,fine,tPen\WObj:=wPaper;
    MoveL Offs(pOrigin,354.34,43.25,6.00),v60,z5,tPen\WObj:=wPaper;
    MoveL Offs(pOrigin,351.29,40.23,6.00),vTravel,z5,tPen\WObj:=wPaper;
    MoveL Offs(pOrigin,351.29,40.23,0.00),v60,z0,tPen\WObj:=wPaper;
    MoveL Offs(pOrigin,344.68,46.84,0.00),v40,z0,tPen\WObj:=wPaper;
    MoveL Offs(pOrigin,345.39,47.00,0.00),v40,z0,tPen\WObj:=wPaper;
    MoveL Offs(pOrigin,346.89,48.50,0.00),v40,z0,tPen\WObj:=wPaper;
    MoveL Offs(pOrigin,347.22,48.78,0.00),v40,z0,tPen\WObj:=wPaper;
    MoveL Offs(pOrigin,329.34,66.66,0.00),v40,z0,tPen\WObj:=wPaper;
    MoveL Offs(pOrigin,328.97,66.43,0.00),v40,z0,tPen\WObj:=wPaper;
    MoveL Offs(pOrigin,327.47,64.92,0.00),v40,z0,tPen\WObj:=wPaper;
    MoveL Offs(pOrigin,326.71,65.69,0.00),v40,z0,tPen\WObj:=wPaper;
    MoveL Offs(pOrigin,329.05,65.69,0.00),v40,z0,tPen\WObj:=wPaper;
    MoveL Offs(pOrigin,329.87,65.83,0.00),v40,z0,tPen\WObj:=wPaper;
    MoveL Offs(pOrigin,328.37,64.33,0.00),v40,z0,tPen\WObj:=wPaper;
    MoveL Offs(pOrigin,329.05,64.63,0.00),v40,z0,tPen\WObj:=wPaper;
    MoveL Offs(pOrigin,330.96,64.63,0.00),v40,z0,tPen\WObj:=wPaper;
    MoveL Offs(pOrigin,330.92,65.38,0.00),v40,z0,tPen\WObj:=wPaper;
    MoveL Offs(pOrigin,329.41,63.88,0.00),v40,z0,tPen\WObj:=wPaper;
    MoveL Offs(pOrigin,328.84,63.22,0.00),v40,z0,tPen\WObj:=wPaper;
    MoveL Offs(pOrigin,333.30,59.19,0.00),v40,z0,tPen\WObj:=wPaper;
    MoveL Offs(pOrigin,336.56,54.72,0.00),v40,z0,tPen\WObj:=wPaper;
    MoveL Offs(pOrigin,338.47,50.90,0.00),v40,z0,tPen\WObj:=wPaper;
    MoveL Offs(pOrigin,339.89,46.22,0.00),v40,z0,tPen\WObj:=wPaper;
    MoveL Offs(pOrigin,340.10,44.31,0.00),v40,fine,tPen\WObj:=wPaper;
    MoveL Offs(pOrigin,340.10,44.31,6.00),v60,z5,tPen\WObj:=wPaper;
    MoveL Offs(pOrigin,340.06,39.52,6.00),vTravel,z5,tPen\WObj:=wPaper;
    MoveL Offs(pOrigin,340.06,39.52,0.00),v60,z0,tPen\WObj:=wPaper;
    MoveL Offs(pOrigin,343.21,36.36,0.00),v40,z0,tPen\WObj:=wPaper;
    MoveL Offs(pOrigin,342.44,35.60,0.00),v40,z0,tPen\WObj:=wPaper;
    MoveL Offs(pOrigin,342.08,34.54,0.00),v40,z0,tPen\WObj:=wPaper;
    MoveL Offs(pOrigin,340.52,32.98,0.00),v40,z0,tPen\WObj:=wPaper;
    MoveL Offs(pOrigin,338.61,32.91,0.00),v40,z0,tPen\WObj:=wPaper;
    MoveL Offs(pOrigin,337.76,34.33,0.00),v40,z0,tPen\WObj:=wPaper;
    MoveL Offs(pOrigin,337.90,36.45,0.00),v40,z0,tPen\WObj:=wPaper;
    MoveL Offs(pOrigin,339.46,38.22,0.00),v40,z0,tPen\WObj:=wPaper;
    MoveL Offs(pOrigin,341.16,38.58,0.00),v40,z0,tPen\WObj:=wPaper;
    MoveL Offs(pOrigin,342.01,38.15,0.00),v40,z0,tPen\WObj:=wPaper;
    MoveL Offs(pOrigin,342.44,37.30,0.00),v40,z0,tPen\WObj:=wPaper;
    MoveL Offs(pOrigin,342.44,35.60,0.00),v40,z0,tPen\WObj:=wPaper;
    MoveL Offs(pOrigin,343.07,35.01,0.00),v40,z0,tPen\WObj:=wPaper;
    MoveL Offs(pOrigin,338.86,39.22,0.00),v40,z0,tPen\WObj:=wPaper;
    MoveL Offs(pOrigin,338.11,38.47,0.00),v40,z0,tPen\WObj:=wPaper;
    MoveL Offs(pOrigin,342.62,33.97,0.00),v40,z0,tPen\WObj:=wPaper;
    MoveL Offs(pOrigin,341.87,33.22,0.00),v40,z0,tPen\WObj:=wPaper;
    MoveL Offs(pOrigin,337.22,37.88,0.00),v40,z0,tPen\WObj:=wPaper;
    MoveL Offs(pOrigin,336.77,36.83,0.00),v40,z0,tPen\WObj:=wPaper;
    MoveL Offs(pOrigin,341.13,32.47,0.00),v40,z0,tPen\WObj:=wPaper;
    MoveL Offs(pOrigin,341.88,31.72,0.00),v40,z0,tPen\WObj:=wPaper;
    MoveL Offs(pOrigin,349.39,24.21,0.00),v40,z0,tPen\WObj:=wPaper;
    MoveL Offs(pOrigin,350.44,24.66,0.00),v40,z0,tPen\WObj:=wPaper;
    MoveL Offs(pOrigin,342.93,32.17,0.00),v40,z0,tPen\WObj:=wPaper;
    MoveL Offs(pOrigin,342.86,31.35,0.00),v40,z0,tPen\WObj:=wPaper;
    MoveL Offs(pOrigin,343.50,31.77,0.00),v40,z0,tPen\WObj:=wPaper;
    MoveL Offs(pOrigin,342.86,31.35,0.00),v40,z0,tPen\WObj:=wPaper;
    MoveL Offs(pOrigin,342.65,30.84,0.00),v40,z0,tPen\WObj:=wPaper;
    MoveL Offs(pOrigin,345.62,30.84,0.00),v40,z0,tPen\WObj:=wPaper;
    MoveL Offs(pOrigin,345.33,31.14,0.00),v40,z0,tPen\WObj:=wPaper;
    MoveL Offs(pOrigin,345.33,32.41,0.00),v40,z0,tPen\WObj:=wPaper;
    MoveL Offs(pOrigin,345.20,32.95,0.00),v40,z0,tPen\WObj:=wPaper;
    MoveL Offs(pOrigin,346.90,32.95,0.00),v40,z0,tPen\WObj:=wPaper;
  ENDPROC

  PROC DrawPart67()
    MoveL Offs(pOrigin,346.69,32.41,0.00),v40,z0,tPen\WObj:=wPaper;
    MoveL Offs(pOrigin,346.90,32.84,0.00),v40,z0,tPen\WObj:=wPaper;
    MoveL Offs(pOrigin,346.69,32.41,0.00),v40,z0,tPen\WObj:=wPaper;
    MoveL Offs(pOrigin,346.26,31.90,0.00),v40,z0,tPen\WObj:=wPaper;
    MoveL Offs(pOrigin,344.14,31.90,0.00),v40,z0,tPen\WObj:=wPaper;
    MoveL Offs(pOrigin,344.14,32.20,0.00),v40,z0,tPen\WObj:=wPaper;
    MoveL Offs(pOrigin,344.99,33.05,0.00),v40,z0,tPen\WObj:=wPaper;
    MoveL Offs(pOrigin,344.14,32.20,0.00),v40,z0,tPen\WObj:=wPaper;
    MoveL Offs(pOrigin,344.27,31.56,0.00),v40,z0,tPen\WObj:=wPaper;
    MoveL Offs(pOrigin,344.27,29.86,0.00),v40,z0,tPen\WObj:=wPaper;
    MoveL Offs(pOrigin,344.99,29.78,0.00),v40,z0,tPen\WObj:=wPaper;
    MoveL Offs(pOrigin,340.10,29.78,0.00),v40,z0,tPen\WObj:=wPaper;
    MoveL Offs(pOrigin,340.05,29.22,0.00),v40,z0,tPen\WObj:=wPaper;
    MoveL Offs(pOrigin,340.05,27.95,0.00),v40,z0,tPen\WObj:=wPaper;
    MoveL Offs(pOrigin,340.31,28.59,0.00),v40,z0,tPen\WObj:=wPaper;
    MoveL Offs(pOrigin,342.01,28.94,0.00),v40,z0,tPen\WObj:=wPaper;
    MoveL Offs(pOrigin,343.29,29.86,0.00),v40,z0,tPen\WObj:=wPaper;
    MoveL Offs(pOrigin,343.21,29.44,0.00),v40,z0,tPen\WObj:=wPaper;
    MoveL Offs(pOrigin,343.21,30.71,0.00),v40,fine,tPen\WObj:=wPaper;
    MoveL Offs(pOrigin,343.21,30.71,6.00),v60,z5,tPen\WObj:=wPaper;
    MoveL Offs(pOrigin,342.01,30.92,6.00),vTravel,z5,tPen\WObj:=wPaper;
    MoveL Offs(pOrigin,342.01,30.92,0.00),v60,z0,tPen\WObj:=wPaper;
    MoveL Offs(pOrigin,342.44,31.14,0.00),v40,z0,tPen\WObj:=wPaper;
    MoveL Offs(pOrigin,342.01,30.92,0.00),v40,fine,tPen\WObj:=wPaper;
    MoveL Offs(pOrigin,342.01,30.92,6.00),v60,z5,tPen\WObj:=wPaper;
    MoveL Offs(pOrigin,340.08,32.03,6.00),vTravel,z5,tPen\WObj:=wPaper;
    MoveL Offs(pOrigin,340.08,32.03,0.00),v60,z0,tPen\WObj:=wPaper;
    MoveL Offs(pOrigin,336.32,35.78,0.00),v40,fine,tPen\WObj:=wPaper;
    MoveL Offs(pOrigin,336.32,35.78,6.00),v60,z5,tPen\WObj:=wPaper;
    MoveL Offs(pOrigin,337.72,36.34,6.00),vTravel,z5,tPen\WObj:=wPaper;
    MoveL Offs(pOrigin,337.72,36.34,0.00),v60,z0,tPen\WObj:=wPaper;
    MoveL Offs(pOrigin,338.62,37.24,0.00),v40,fine,tPen\WObj:=wPaper;
    MoveL Offs(pOrigin,338.62,37.24,6.00),v60,z5,tPen\WObj:=wPaper;
    MoveL Offs(pOrigin,340.10,35.39,6.00),vTravel,z5,tPen\WObj:=wPaper;
    MoveL Offs(pOrigin,340.10,35.39,0.00),v60,z0,tPen\WObj:=wPaper;
    MoveL Offs(pOrigin,340.74,36.03,0.00),v40,fine,tPen\WObj:=wPaper;
    MoveL Offs(pOrigin,340.74,36.03,6.00),v60,z5,tPen\WObj:=wPaper;
    MoveL Offs(pOrigin,343.52,33.07,6.00),vTravel,z5,tPen\WObj:=wPaper;
    MoveL Offs(pOrigin,343.52,33.07,0.00),v60,z0,tPen\WObj:=wPaper;
    MoveL Offs(pOrigin,351.49,25.10,0.00),v40,fine,tPen\WObj:=wPaper;
    MoveL Offs(pOrigin,351.49,25.10,6.00),v60,z5,tPen\WObj:=wPaper;
    MoveL Offs(pOrigin,350.51,26.62,6.00),vTravel,z5,tPen\WObj:=wPaper;
    MoveL Offs(pOrigin,350.51,26.62,0.00),v60,z0,tPen\WObj:=wPaper;
    MoveL Offs(pOrigin,352.85,26.62,0.00),v40,fine,tPen\WObj:=wPaper;
    MoveL Offs(pOrigin,352.85,26.62,6.00),v60,z5,tPen\WObj:=wPaper;
    MoveL Offs(pOrigin,349.23,28.85,6.00),vTravel,z5,tPen\WObj:=wPaper;
    MoveL Offs(pOrigin,349.23,28.85,0.00),v60,z0,tPen\WObj:=wPaper;
    MoveL Offs(pOrigin,344.42,33.66,0.00),v40,z0,tPen\WObj:=wPaper;
    MoveL Offs(pOrigin,345.41,33.69,0.00),v40,z0,tPen\WObj:=wPaper;
    MoveL Offs(pOrigin,345.62,34.11,0.00),v40,z0,tPen\WObj:=wPaper;
    MoveL Offs(pOrigin,345.41,33.69,0.00),v40,z0,tPen\WObj:=wPaper;
    MoveL Offs(pOrigin,346.05,34.01,0.00),v40,z0,tPen\WObj:=wPaper;
    MoveL Offs(pOrigin,347.33,34.01,0.00),v40,z0,tPen\WObj:=wPaper;
    MoveL Offs(pOrigin,347.75,35.06,0.00),v40,z0,tPen\WObj:=wPaper;
    MoveL Offs(pOrigin,346.69,35.06,0.00),v40,z0,tPen\WObj:=wPaper;
    MoveL Offs(pOrigin,347.11,36.12,0.00),v40,z0,tPen\WObj:=wPaper;
    MoveL Offs(pOrigin,348.17,36.12,0.00),v40,fine,tPen\WObj:=wPaper;
    MoveL Offs(pOrigin,348.17,36.12,6.00),v60,z5,tPen\WObj:=wPaper;
    MoveL Offs(pOrigin,345.91,36.65,6.00),vTravel,z5,tPen\WObj:=wPaper;
    MoveL Offs(pOrigin,345.91,36.65,0.00),v60,z0,tPen\WObj:=wPaper;
    MoveL Offs(pOrigin,351.02,31.54,0.00),v40,fine,tPen\WObj:=wPaper;
    MoveL Offs(pOrigin,351.02,31.54,6.00),v60,z5,tPen\WObj:=wPaper;
    MoveL Offs(pOrigin,352.36,33.19,6.00),vTravel,z5,tPen\WObj:=wPaper;
    MoveL Offs(pOrigin,352.36,33.19,0.00),v60,z0,tPen\WObj:=wPaper;
    MoveL Offs(pOrigin,346.50,39.05,0.00),v40,fine,tPen\WObj:=wPaper;
    MoveL Offs(pOrigin,346.50,39.05,6.00),v60,z5,tPen\WObj:=wPaper;
    MoveL Offs(pOrigin,346.79,41.74,6.00),vTravel,z5,tPen\WObj:=wPaper;
    MoveL Offs(pOrigin,346.79,41.74,0.00),v60,z0,tPen\WObj:=wPaper;
    MoveL Offs(pOrigin,351.75,36.79,0.00),v40,z0,tPen\WObj:=wPaper;
    MoveL Offs(pOrigin,351.05,36.23,0.00),v40,z0,tPen\WObj:=wPaper;
    MoveL Offs(pOrigin,348.65,33.83,0.00),v40,fine,tPen\WObj:=wPaper;
    MoveL Offs(pOrigin,348.65,33.83,6.00),v60,z5,tPen\WObj:=wPaper;
    MoveL Offs(pOrigin,349.24,30.29,6.00),vTravel,z5,tPen\WObj:=wPaper;
    MoveL Offs(pOrigin,349.24,30.29,0.00),v60,z0,tPen\WObj:=wPaper;
    MoveL Offs(pOrigin,349.45,30.71,0.00),v40,z0,tPen\WObj:=wPaper;
    MoveL Offs(pOrigin,349.24,30.29,0.00),v40,z0,tPen\WObj:=wPaper;
    MoveL Offs(pOrigin,349.38,30.09,0.00),v40,z0,tPen\WObj:=wPaper;
    MoveL Offs(pOrigin,343.07,23.78,0.00),v40,z0,tPen\WObj:=wPaper;
    MoveL Offs(pOrigin,342.95,23.18,0.00),v40,z0,tPen\WObj:=wPaper;
    MoveL Offs(pOrigin,336.34,29.79,0.00),v40,z0,tPen\WObj:=wPaper;
    MoveL Offs(pOrigin,336.80,29.45,0.00),v40,z0,tPen\WObj:=wPaper;
    MoveL Offs(pOrigin,333.64,26.29,0.00),v40,z0,tPen\WObj:=wPaper;
    MoveL Offs(pOrigin,333.94,26.62,0.00),v40,z0,tPen\WObj:=wPaper;
    MoveL Offs(pOrigin,337.55,26.62,0.00),v40,fine,tPen\WObj:=wPaper;
    MoveL Offs(pOrigin,337.55,26.62,6.00),v60,z5,tPen\WObj:=wPaper;
    MoveL Offs(pOrigin,336.78,24.96,6.00),vTravel,z5,tPen\WObj:=wPaper;
    MoveL Offs(pOrigin,336.78,24.96,0.00),v60,z0,tPen\WObj:=wPaper;
    MoveL Offs(pOrigin,351.06,39.23,0.00),v40,z0,tPen\WObj:=wPaper;
    MoveL Offs(pOrigin,351.75,38.28,0.00),v40,z0,tPen\WObj:=wPaper;
    MoveL Offs(pOrigin,346.34,43.69,0.00),v40,fine,tPen\WObj:=wPaper;
    MoveL Offs(pOrigin,346.34,43.69,6.00),v60,z5,tPen\WObj:=wPaper;
    MoveL Offs(pOrigin,346.58,45.21,6.00),vTravel,z5,tPen\WObj:=wPaper;
    MoveL Offs(pOrigin,346.58,45.21,0.00),v60,z0,tPen\WObj:=wPaper;
    MoveL Offs(pOrigin,348.09,46.71,0.00),v40,z0,tPen\WObj:=wPaper;
    MoveL Offs(pOrigin,347.75,46.44,0.00),v40,z0,tPen\WObj:=wPaper;
    MoveL Offs(pOrigin,347.33,47.08,0.00),v40,z0,tPen\WObj:=wPaper;
    MoveL Offs(pOrigin,347.75,46.44,0.00),v40,z0,tPen\WObj:=wPaper;
    MoveL Offs(pOrigin,347.33,46.68,0.00),v40,z0,tPen\WObj:=wPaper;
    MoveL Offs(pOrigin,346.26,46.68,0.00),v40,z0,tPen\WObj:=wPaper;
    MoveL Offs(pOrigin,346.05,46.44,0.00),v40,z0,tPen\WObj:=wPaper;
    MoveL Offs(pOrigin,345.84,46.86,0.00),v40,z0,tPen\WObj:=wPaper;
    MoveL Offs(pOrigin,346.05,46.44,0.00),v40,z0,tPen\WObj:=wPaper;
    MoveL Offs(pOrigin,345.99,46.11,0.00),v40,z0,tPen\WObj:=wPaper;
    MoveL Offs(pOrigin,347.49,47.61,0.00),v40,z0,tPen\WObj:=wPaper;
    MoveL Offs(pOrigin,347.11,47.50,0.00),v40,z0,tPen\WObj:=wPaper;
    MoveL Offs(pOrigin,346.90,47.92,0.00),v40,z0,tPen\WObj:=wPaper;
    MoveL Offs(pOrigin,347.11,47.50,0.00),v40,z0,tPen\WObj:=wPaper;
    MoveL Offs(pOrigin,346.69,47.74,0.00),v40,z0,tPen\WObj:=wPaper;
    MoveL Offs(pOrigin,345.62,47.74,0.00),v40,z0,tPen\WObj:=wPaper;
    MoveL Offs(pOrigin,345.41,47.50,0.00),v40,z0,tPen\WObj:=wPaper;
    MoveL Offs(pOrigin,345.20,47.92,0.00),v40,z0,tPen\WObj:=wPaper;
    MoveL Offs(pOrigin,345.41,47.50,0.00),v40,z0,tPen\WObj:=wPaper;
    MoveL Offs(pOrigin,344.94,48.05,0.00),v40,z0,tPen\WObj:=wPaper;
    MoveL Offs(pOrigin,346.30,49.40,0.00),v40,z0,tPen\WObj:=wPaper;
    MoveL Offs(pOrigin,346.05,48.79,0.00),v40,z0,tPen\WObj:=wPaper;
    MoveL Offs(pOrigin,344.99,48.79,0.00),v40,z0,tPen\WObj:=wPaper;
    MoveL Offs(pOrigin,344.35,48.95,0.00),v40,z0,tPen\WObj:=wPaper;
    MoveL Offs(pOrigin,345.85,50.45,0.00),v40,z0,tPen\WObj:=wPaper;
    MoveL Offs(pOrigin,345.41,50.26,0.00),v40,z0,tPen\WObj:=wPaper;
    MoveL Offs(pOrigin,344.99,50.90,0.00),v40,z0,tPen\WObj:=wPaper;
  ENDPROC

  PROC DrawPart68()
    MoveL Offs(pOrigin,345.41,50.26,0.00),v40,z0,tPen\WObj:=wPaper;
    MoveL Offs(pOrigin,345.41,49.85,0.00),v40,z0,tPen\WObj:=wPaper;
    MoveL Offs(pOrigin,344.35,49.85,0.00),v40,z0,tPen\WObj:=wPaper;
    MoveL Offs(pOrigin,343.75,49.84,0.00),v40,z0,tPen\WObj:=wPaper;
    MoveL Offs(pOrigin,345.25,51.35,0.00),v40,z0,tPen\WObj:=wPaper;
    MoveL Offs(pOrigin,345.71,51.78,0.00),v40,z0,tPen\WObj:=wPaper;
    MoveL Offs(pOrigin,331.89,65.61,0.00),v40,z0,tPen\WObj:=wPaper;
    MoveL Offs(pOrigin,331.81,64.79,0.00),v40,z0,tPen\WObj:=wPaper;
    MoveL Offs(pOrigin,330.31,63.28,0.00),v40,z0,tPen\WObj:=wPaper;
    MoveL Offs(pOrigin,330.75,63.58,0.00),v40,z0,tPen\WObj:=wPaper;
    MoveL Offs(pOrigin,332.66,63.58,0.00),v40,z0,tPen\WObj:=wPaper;
    MoveL Offs(pOrigin,332.71,64.19,0.00),v40,z0,tPen\WObj:=wPaper;
    MoveL Offs(pOrigin,331.21,62.69,0.00),v40,z0,tPen\WObj:=wPaper;
    MoveL Offs(pOrigin,332.11,62.09,0.00),v40,z0,tPen\WObj:=wPaper;
    MoveL Offs(pOrigin,333.61,63.59,0.00),v40,z0,tPen\WObj:=wPaper;
    MoveL Offs(pOrigin,334.50,63.00,0.00),v40,z0,tPen\WObj:=wPaper;
    MoveL Offs(pOrigin,333.00,61.49,0.00),v40,z0,tPen\WObj:=wPaper;
    MoveL Offs(pOrigin,333.72,61.46,0.00),v40,z0,tPen\WObj:=wPaper;
    MoveL Offs(pOrigin,335.64,61.46,0.00),v40,z0,tPen\WObj:=wPaper;
    MoveL Offs(pOrigin,336.15,61.65,0.00),v40,z0,tPen\WObj:=wPaper;
    MoveL Offs(pOrigin,334.65,60.15,0.00),v40,z0,tPen\WObj:=wPaper;
    MoveL Offs(pOrigin,335.00,60.25,0.00),v40,z0,tPen\WObj:=wPaper;
    MoveL Offs(pOrigin,334.58,60.67,0.00),v40,z0,tPen\WObj:=wPaper;
    MoveL Offs(pOrigin,335.00,60.25,0.00),v40,z0,tPen\WObj:=wPaper;
    MoveL Offs(pOrigin,335.21,60.41,0.00),v40,z0,tPen\WObj:=wPaper;
    MoveL Offs(pOrigin,336.70,60.41,0.00),v40,z0,tPen\WObj:=wPaper;
    MoveL Offs(pOrigin,336.91,60.46,0.00),v40,z0,tPen\WObj:=wPaper;
    MoveL Offs(pOrigin,335.85,61.53,0.00),v40,z0,tPen\WObj:=wPaper;
    MoveL Offs(pOrigin,336.91,60.46,0.00),v40,z0,tPen\WObj:=wPaper;
    MoveL Offs(pOrigin,337.05,61.06,0.00),v40,z0,tPen\WObj:=wPaper;
    MoveL Offs(pOrigin,335.54,59.56,0.00),v40,fine,tPen\WObj:=wPaper;
    MoveL Offs(pOrigin,335.54,59.56,6.00),v60,z5,tPen\WObj:=wPaper;
    MoveL Offs(pOrigin,333.75,60.75,6.00),vTravel,z5,tPen\WObj:=wPaper;
    MoveL Offs(pOrigin,333.75,60.75,0.00),v60,z0,tPen\WObj:=wPaper;
    MoveL Offs(pOrigin,335.40,62.40,0.00),v40,z0,tPen\WObj:=wPaper;
    MoveL Offs(pOrigin,335.21,61.95,0.00),v40,z0,tPen\WObj:=wPaper;
    MoveL Offs(pOrigin,334.79,62.38,0.00),v40,z0,tPen\WObj:=wPaper;
    MoveL Offs(pOrigin,335.21,61.95,0.00),v40,fine,tPen\WObj:=wPaper;
    MoveL Offs(pOrigin,335.21,61.95,6.00),v60,z5,tPen\WObj:=wPaper;
    MoveL Offs(pOrigin,334.15,62.52,6.00),vTravel,z5,tPen\WObj:=wPaper;
    MoveL Offs(pOrigin,334.15,62.52,0.00),v60,z0,tPen\WObj:=wPaper;
    MoveL Offs(pOrigin,332.45,62.52,0.00),v40,fine,tPen\WObj:=wPaper;
    MoveL Offs(pOrigin,332.45,62.52,6.00),v60,z5,tPen\WObj:=wPaper;
    MoveL Offs(pOrigin,327.85,63.67,6.00),vTravel,z5,tPen\WObj:=wPaper;
    MoveL Offs(pOrigin,327.85,63.67,0.00),v60,z0,tPen\WObj:=wPaper;
    MoveL Offs(pOrigin,318.98,72.54,0.00),v40,fine,tPen\WObj:=wPaper;
    MoveL Offs(pOrigin,318.98,72.54,6.00),v60,z5,tPen\WObj:=wPaper;
    MoveL Offs(pOrigin,316.74,71.80,6.00),vTravel,z5,tPen\WObj:=wPaper;
    MoveL Offs(pOrigin,316.74,71.80,0.00),v60,z0,tPen\WObj:=wPaper;
    MoveL Offs(pOrigin,322.75,65.79,0.00),v40,fine,tPen\WObj:=wPaper;
    MoveL Offs(pOrigin,322.75,65.79,6.00),v60,z5,tPen\WObj:=wPaper;
    MoveL Offs(pOrigin,319.30,66.25,6.00),vTravel,z5,tPen\WObj:=wPaper;
    MoveL Offs(pOrigin,319.30,66.25,0.00),v60,z0,tPen\WObj:=wPaper;
    MoveL Offs(pOrigin,314.50,71.05,0.00),v40,fine,tPen\WObj:=wPaper;
    MoveL Offs(pOrigin,314.50,71.05,6.00),v60,z5,tPen\WObj:=wPaper;
    MoveL Offs(pOrigin,315.03,62.94,6.00),vTravel,z5,tPen\WObj:=wPaper;
    MoveL Offs(pOrigin,315.03,62.94,0.00),v60,z0,tPen\WObj:=wPaper;
    MoveL Offs(pOrigin,311.88,59.78,0.00),v40,z0,tPen\WObj:=wPaper;
    MoveL Offs(pOrigin,311.39,59.23,0.00),v40,z0,tPen\WObj:=wPaper;
    MoveL Offs(pOrigin,303.87,66.74,0.00),v40,fine,tPen\WObj:=wPaper;
    MoveL Offs(pOrigin,303.87,66.74,6.00),v60,z5,tPen\WObj:=wPaper;
    MoveL Offs(pOrigin,302.68,66.45,6.00),vTravel,z5,tPen\WObj:=wPaper;
    MoveL Offs(pOrigin,302.68,66.45,0.00),v60,z0,tPen\WObj:=wPaper;
    MoveL Offs(pOrigin,310.04,59.08,0.00),v40,fine,tPen\WObj:=wPaper;
    MoveL Offs(pOrigin,310.04,59.08,6.00),v60,z5,tPen\WObj:=wPaper;
    MoveL Offs(pOrigin,309.42,60.68,6.00),vTravel,z5,tPen\WObj:=wPaper;
    MoveL Offs(pOrigin,309.42,60.68,0.00),v60,z0,tPen\WObj:=wPaper;
    MoveL Offs(pOrigin,309.42,62.16,0.00),v40,fine,tPen\WObj:=wPaper;
    MoveL Offs(pOrigin,309.42,62.16,6.00),v60,z5,tPen\WObj:=wPaper;
    MoveL Offs(pOrigin,308.23,62.52,6.00),vTravel,z5,tPen\WObj:=wPaper;
    MoveL Offs(pOrigin,308.23,62.52,0.00),v60,z0,tPen\WObj:=wPaper;
    MoveL Offs(pOrigin,314.39,62.52,0.00),v40,z0,tPen\WObj:=wPaper;
    MoveL Offs(pOrigin,314.70,61.95,0.00),v40,z0,tPen\WObj:=wPaper;
    MoveL Offs(pOrigin,314.70,60.68,0.00),v40,z0,tPen\WObj:=wPaper;
    MoveL Offs(pOrigin,313.65,60.89,0.00),v40,z0,tPen\WObj:=wPaper;
    MoveL Offs(pOrigin,313.65,62.16,0.00),v40,fine,tPen\WObj:=wPaper;
    MoveL Offs(pOrigin,313.65,62.16,6.00),v60,z5,tPen\WObj:=wPaper;
    MoveL Offs(pOrigin,315.93,62.34,6.00),vTravel,z5,tPen\WObj:=wPaper;
    MoveL Offs(pOrigin,315.93,62.34,0.00),v60,z0,tPen\WObj:=wPaper;
    MoveL Offs(pOrigin,313.37,59.79,0.00),v40,z0,tPen\WObj:=wPaper;
    MoveL Offs(pOrigin,313.18,58.92,0.00),v40,z0,tPen\WObj:=wPaper;
    MoveL Offs(pOrigin,305.07,67.04,0.00),v40,fine,tPen\WObj:=wPaper;
    MoveL Offs(pOrigin,305.07,67.04,6.00),v60,z5,tPen\WObj:=wPaper;
    MoveL Offs(pOrigin,302.49,63.22,6.00),vTravel,z5,tPen\WObj:=wPaper;
    MoveL Offs(pOrigin,302.49,63.22,0.00),v60,z0,tPen\WObj:=wPaper;
    MoveL Offs(pOrigin,306.74,64.07,0.00),v40,z0,tPen\WObj:=wPaper;
    MoveL Offs(pOrigin,310.14,64.07,0.00),v40,z0,tPen\WObj:=wPaper;
    MoveL Offs(pOrigin,314.39,62.87,0.00),v40,z0,tPen\WObj:=wPaper;
    MoveL Offs(pOrigin,317.43,60.96,0.00),v40,z0,tPen\WObj:=wPaper;
    MoveL Offs(pOrigin,317.15,61.10,0.00),v40,z0,tPen\WObj:=wPaper;
    MoveL Offs(pOrigin,316.73,61.31,0.00),v40,z0,tPen\WObj:=wPaper;
    MoveL Offs(pOrigin,316.30,61.74,0.00),v40,z0,tPen\WObj:=wPaper;
    MoveL Offs(pOrigin,316.73,61.31,0.00),v40,z0,tPen\WObj:=wPaper;
    MoveL Offs(pOrigin,316.82,61.74,0.00),v40,z0,tPen\WObj:=wPaper;
    MoveL Offs(pOrigin,314.42,59.34,0.00),v40,fine,tPen\WObj:=wPaper;
    MoveL Offs(pOrigin,314.42,59.34,6.00),v60,z5,tPen\WObj:=wPaper;
    MoveL Offs(pOrigin,315.62,59.04,6.00),vTravel,z5,tPen\WObj:=wPaper;
    MoveL Offs(pOrigin,315.62,59.04,0.00),v60,z0,tPen\WObj:=wPaper;
    MoveL Offs(pOrigin,317.72,61.15,0.00),v40,z0,tPen\WObj:=wPaper;
    MoveL Offs(pOrigin,318.12,61.46,0.00),v40,z0,tPen\WObj:=wPaper;
    MoveL Offs(pOrigin,319.62,59.95,0.00),v40,z0,tPen\WObj:=wPaper;
    MoveL Offs(pOrigin,319.22,59.65,0.00),v40,z0,tPen\WObj:=wPaper;
    MoveL Offs(pOrigin,317.11,57.55,0.00),v40,z0,tPen\WObj:=wPaper;
    MoveL Offs(pOrigin,317.58,57.28,0.00),v40,z0,tPen\WObj:=wPaper;
    MoveL Offs(pOrigin,316.94,57.91,0.00),v40,z0,tPen\WObj:=wPaper;
    MoveL Offs(pOrigin,317.58,57.28,0.00),v40,z0,tPen\WObj:=wPaper;
    MoveL Offs(pOrigin,317.71,56.65,0.00),v40,z0,tPen\WObj:=wPaper;
    MoveL Offs(pOrigin,319.81,58.76,0.00),v40,z0,tPen\WObj:=wPaper;
    MoveL Offs(pOrigin,319.70,58.76,0.00),v40,z0,tPen\WObj:=wPaper;
    MoveL Offs(pOrigin,319.91,58.34,0.00),v40,z0,tPen\WObj:=wPaper;
    MoveL Offs(pOrigin,319.70,58.76,0.00),v40,z0,tPen\WObj:=wPaper;
    MoveL Offs(pOrigin,319.49,58.30,0.00),v40,z0,tPen\WObj:=wPaper;
    MoveL Offs(pOrigin,318.00,58.30,0.00),v40,fine,tPen\WObj:=wPaper;
    MoveL Offs(pOrigin,318.00,58.30,6.00),v60,z5,tPen\WObj:=wPaper;
    MoveL Offs(pOrigin,318.64,59.35,6.00),vTravel,z5,tPen\WObj:=wPaper;
    MoveL Offs(pOrigin,318.64,59.35,0.00),v60,z0,tPen\WObj:=wPaper;
    MoveL Offs(pOrigin,317.15,59.35,0.00),v40,fine,tPen\WObj:=wPaper;
    MoveL Offs(pOrigin,317.15,59.35,6.00),v60,z5,tPen\WObj:=wPaper;
    MoveL Offs(pOrigin,316.09,58.76,6.00),vTravel,z5,tPen\WObj:=wPaper;
    MoveL Offs(pOrigin,316.09,58.76,0.00),v60,z0,tPen\WObj:=wPaper;
  ENDPROC

  PROC DrawPart69()
    MoveL Offs(pOrigin,315.66,59.19,0.00),v40,z0,tPen\WObj:=wPaper;
    MoveL Offs(pOrigin,316.09,58.76,0.00),v40,z0,tPen\WObj:=wPaper;
    MoveL Offs(pOrigin,316.36,58.30,0.00),v40,z0,tPen\WObj:=wPaper;
    MoveL Offs(pOrigin,318.47,60.40,0.00),v40,z0,tPen\WObj:=wPaper;
    MoveL Offs(pOrigin,318.85,59.61,0.00),v40,z0,tPen\WObj:=wPaper;
    MoveL Offs(pOrigin,318.64,60.04,0.00),v40,z0,tPen\WObj:=wPaper;
    MoveL Offs(pOrigin,318.85,59.61,0.00),v40,fine,tPen\WObj:=wPaper;
    MoveL Offs(pOrigin,318.85,59.61,6.00),v60,z5,tPen\WObj:=wPaper;
    MoveL Offs(pOrigin,316.30,61.46,6.00),vTravel,z5,tPen\WObj:=wPaper;
    MoveL Offs(pOrigin,316.30,61.46,0.00),v60,z0,tPen\WObj:=wPaper;
    MoveL Offs(pOrigin,307.59,61.46,0.00),v40,fine,tPen\WObj:=wPaper;
    MoveL Offs(pOrigin,307.59,61.46,6.00),v60,z5,tPen\WObj:=wPaper;
    MoveL Offs(pOrigin,304.40,56.21,6.00),vTravel,z5,tPen\WObj:=wPaper;
    MoveL Offs(pOrigin,304.40,56.21,0.00),v60,z0,tPen\WObj:=wPaper;
    MoveL Offs(pOrigin,307.73,51.33,0.00),v40,z0,tPen\WObj:=wPaper;
    MoveL Offs(pOrigin,308.44,49.62,0.00),v40,z0,tPen\WObj:=wPaper;
    MoveL Offs(pOrigin,308.44,48.78,0.00),v40,fine,tPen\WObj:=wPaper;
    MoveL Offs(pOrigin,308.44,48.78,6.00),v60,z5,tPen\WObj:=wPaper;
    MoveL Offs(pOrigin,305.89,45.16,6.00),vTravel,z5,tPen\WObj:=wPaper;
    MoveL Offs(pOrigin,305.89,45.16,0.00),v60,z0,tPen\WObj:=wPaper;
    MoveL Offs(pOrigin,305.89,46.44,0.00),v40,z0,tPen\WObj:=wPaper;
    MoveL Offs(pOrigin,304.26,50.90,0.00),v40,z0,tPen\WObj:=wPaper;
    MoveL Offs(pOrigin,302.63,53.88,0.00),v40,z0,tPen\WObj:=wPaper;
    MoveL Offs(pOrigin,300.15,57.06,0.00),v40,fine,tPen\WObj:=wPaper;
    MoveL Offs(pOrigin,300.15,57.06,6.00),v60,z5,tPen\WObj:=wPaper;
    MoveL Offs(pOrigin,300.90,59.26,6.00),vTravel,z5,tPen\WObj:=wPaper;
    MoveL Offs(pOrigin,300.90,59.26,0.00),v60,z0,tPen\WObj:=wPaper;
    MoveL Offs(pOrigin,293.24,66.92,0.00),v40,fine,tPen\WObj:=wPaper;
    MoveL Offs(pOrigin,293.24,66.92,6.00),v60,z5,tPen\WObj:=wPaper;
    MoveL Offs(pOrigin,292.94,65.73,6.00),vTravel,z5,tPen\WObj:=wPaper;
    MoveL Offs(pOrigin,292.94,65.73,0.00),v60,z0,tPen\WObj:=wPaper;
    MoveL Offs(pOrigin,298.95,59.72,0.00),v40,fine,tPen\WObj:=wPaper;
    MoveL Offs(pOrigin,298.95,59.72,6.00),v60,z5,tPen\WObj:=wPaper;
    MoveL Offs(pOrigin,296.70,60.47,6.00),vTravel,z5,tPen\WObj:=wPaper;
    MoveL Offs(pOrigin,296.70,60.47,0.00),v60,z0,tPen\WObj:=wPaper;
    MoveL Offs(pOrigin,290.54,66.63,0.00),v40,z0,tPen\WObj:=wPaper;
    MoveL Offs(pOrigin,290.02,66.31,0.00),v40,z0,tPen\WObj:=wPaper;
    MoveL Offs(pOrigin,288.52,64.80,0.00),v40,z0,tPen\WObj:=wPaper;
    MoveL Offs(pOrigin,289.52,64.63,0.00),v40,z0,tPen\WObj:=wPaper;
    MoveL Offs(pOrigin,291.86,64.63,0.00),v40,z0,tPen\WObj:=wPaper;
    MoveL Offs(pOrigin,291.97,65.26,0.00),v40,z0,tPen\WObj:=wPaper;
    MoveL Offs(pOrigin,290.47,63.76,0.00),v40,z0,tPen\WObj:=wPaper;
    MoveL Offs(pOrigin,291.36,63.16,0.00),v40,z0,tPen\WObj:=wPaper;
    MoveL Offs(pOrigin,293.02,64.82,0.00),v40,fine,tPen\WObj:=wPaper;
    MoveL Offs(pOrigin,293.02,64.82,6.00),v60,z5,tPen\WObj:=wPaper;
    MoveL Offs(pOrigin,294.36,64.67,6.00),vTravel,z5,tPen\WObj:=wPaper;
    MoveL Offs(pOrigin,294.36,64.67,0.00),v60,z0,tPen\WObj:=wPaper;
    MoveL Offs(pOrigin,292.41,62.72,0.00),v40,z0,tPen\WObj:=wPaper;
    MoveL Offs(pOrigin,292.35,61.83,0.00),v40,z0,tPen\WObj:=wPaper;
    MoveL Offs(pOrigin,284.09,70.10,0.00),v40,z0,tPen\WObj:=wPaper;
    MoveL Offs(pOrigin,283.34,69.35,0.00),v40,z0,tPen\WObj:=wPaper;
    MoveL Offs(pOrigin,289.05,63.64,0.00),v40,z0,tPen\WObj:=wPaper;
    MoveL Offs(pOrigin,289.42,64.21,0.00),v40,z0,tPen\WObj:=wPaper;
    MoveL Offs(pOrigin,290.92,65.71,0.00),v40,z0,tPen\WObj:=wPaper;
    MoveL Offs(pOrigin,290.59,65.56,0.00),v40,z0,tPen\WObj:=wPaper;
    MoveL Offs(pOrigin,292.92,64.36,0.00),v40,z0,tPen\WObj:=wPaper;
    MoveL Offs(pOrigin,294.62,64.07,0.00),v40,z0,tPen\WObj:=wPaper;
    MoveL Offs(pOrigin,294.62,63.58,0.00),v40,z0,tPen\WObj:=wPaper;
    MoveL Offs(pOrigin,291.65,63.58,0.00),v40,fine,tPen\WObj:=wPaper;
    MoveL Offs(pOrigin,291.65,63.58,6.00),v60,z5,tPen\WObj:=wPaper;
    MoveL Offs(pOrigin,291.23,65.35,6.00),vTravel,z5,tPen\WObj:=wPaper;
    MoveL Offs(pOrigin,291.23,65.35,0.00),v60,z0,tPen\WObj:=wPaper;
    MoveL Offs(pOrigin,291.65,65.14,0.00),v40,z0,tPen\WObj:=wPaper;
    MoveL Offs(pOrigin,291.23,65.35,0.00),v40,fine,tPen\WObj:=wPaper;
    MoveL Offs(pOrigin,291.23,65.35,6.00),v60,z5,tPen\WObj:=wPaper;
    MoveL Offs(pOrigin,289.95,65.78,6.00),vTravel,z5,tPen\WObj:=wPaper;
    MoveL Offs(pOrigin,289.95,65.78,0.00),v60,z0,tPen\WObj:=wPaper;
    MoveL Offs(pOrigin,286.76,67.69,0.00),v40,z0,tPen\WObj:=wPaper;
    MoveL Offs(pOrigin,286.55,69.81,0.00),v40,z0,tPen\WObj:=wPaper;
    MoveL Offs(pOrigin,288.25,80.44,0.00),v40,z0,tPen\WObj:=wPaper;
    MoveL Offs(pOrigin,291.30,93.82,0.00),v40,z0,tPen\WObj:=wPaper;
    MoveL Offs(pOrigin,292.08,94.46,0.00),v40,z0,tPen\WObj:=wPaper;
    MoveL Offs(pOrigin,291.65,94.20,0.00),v40,z0,tPen\WObj:=wPaper;
    MoveL Offs(pOrigin,289.95,94.20,0.00),v40,z0,tPen\WObj:=wPaper;
    MoveL Offs(pOrigin,289.21,93.87,0.00),v40,z0,tPen\WObj:=wPaper;
    MoveL Offs(pOrigin,293.12,97.77,0.00),v40,z0,tPen\WObj:=wPaper;
    MoveL Offs(pOrigin,293.44,98.08,0.00),v40,z0,tPen\WObj:=wPaper;
    MoveL Offs(pOrigin,290.59,100.94,0.00),v40,z0,tPen\WObj:=wPaper;
    MoveL Offs(pOrigin,291.65,100.54,0.00),v40,z0,tPen\WObj:=wPaper;
    MoveL Offs(pOrigin,292.92,100.54,0.00),v40,z0,tPen\WObj:=wPaper;
    MoveL Offs(pOrigin,293.43,101.07,0.00),v40,z0,tPen\WObj:=wPaper;
    MoveL Offs(pOrigin,290.12,97.76,0.00),v40,z0,tPen\WObj:=wPaper;
    MoveL Offs(pOrigin,289.55,97.49,0.00),v40,z0,tPen\WObj:=wPaper;
    MoveL Offs(pOrigin,293.30,93.74,0.00),v40,z0,tPen\WObj:=wPaper;
    MoveL Offs(pOrigin,292.51,94.18,0.00),v40,z0,tPen\WObj:=wPaper;
    MoveL Offs(pOrigin,288.45,90.12,0.00),v40,z0,tPen\WObj:=wPaper;
    MoveL Offs(pOrigin,287.92,90.16,0.00),v40,z0,tPen\WObj:=wPaper;
    MoveL Offs(pOrigin,293.03,85.05,0.00),v40,fine,tPen\WObj:=wPaper;
    MoveL Offs(pOrigin,293.03,85.05,6.00),v60,z5,tPen\WObj:=wPaper;
    MoveL Offs(pOrigin,293.03,86.55,6.00),vTravel,z5,tPen\WObj:=wPaper;
    MoveL Offs(pOrigin,293.03,86.55,0.00),v60,z0,tPen\WObj:=wPaper;
    MoveL Offs(pOrigin,288.07,91.51,0.00),v40,z0,tPen\WObj:=wPaper;
    MoveL Offs(pOrigin,288.91,92.07,0.00),v40,z0,tPen\WObj:=wPaper;
    MoveL Offs(pOrigin,292.66,95.82,0.00),v40,z0,tPen\WObj:=wPaper;
    MoveL Offs(pOrigin,292.29,96.31,0.00),v40,z0,tPen\WObj:=wPaper;
    MoveL Offs(pOrigin,290.59,96.31,0.00),v40,z0,tPen\WObj:=wPaper;
    MoveL Offs(pOrigin,289.97,96.12,0.00),v40,z0,tPen\WObj:=wPaper;
    MoveL Offs(pOrigin,293.42,99.57,0.00),v40,z0,tPen\WObj:=wPaper;
    MoveL Offs(pOrigin,293.74,99.28,0.00),v40,z0,tPen\WObj:=wPaper;
    MoveL Offs(pOrigin,290.88,102.13,0.00),v40,z0,tPen\WObj:=wPaper;
    MoveL Offs(pOrigin,291.33,101.96,0.00),v40,z0,tPen\WObj:=wPaper;
    MoveL Offs(pOrigin,295.99,106.62,0.00),v40,z0,tPen\WObj:=wPaper;
    MoveL Offs(pOrigin,296.11,105.94,0.00),v40,z0,tPen\WObj:=wPaper;
    MoveL Offs(pOrigin,295.26,106.15,0.00),v40,z0,tPen\WObj:=wPaper;
    MoveL Offs(pOrigin,295.05,107.43,0.00),v40,z0,tPen\WObj:=wPaper;
    MoveL Offs(pOrigin,297.53,115.50,0.00),v40,z0,tPen\WObj:=wPaper;
    MoveL Offs(pOrigin,298.02,116.07,0.00),v40,z0,tPen\WObj:=wPaper;
    MoveL Offs(pOrigin,342.86,128.89,0.00),v40,z0,tPen\WObj:=wPaper;
    MoveL Offs(pOrigin,344.35,129.10,0.00),v40,z0,tPen\WObj:=wPaper;
    MoveL Offs(pOrigin,344.56,128.89,0.00),v40,z0,tPen\WObj:=wPaper;
    MoveL Offs(pOrigin,344.77,119.75,0.00),v40,z0,tPen\WObj:=wPaper;
    MoveL Offs(pOrigin,344.49,119.11,0.00),v40,z0,tPen\WObj:=wPaper;
    MoveL Offs(pOrigin,343.71,118.62,0.00),v40,z0,tPen\WObj:=wPaper;
    MoveL Offs(pOrigin,324.38,112.95,0.00),v40,z0,tPen\WObj:=wPaper;
    MoveL Offs(pOrigin,297.17,106.15,0.00),v40,z0,tPen\WObj:=wPaper;
    MoveL Offs(pOrigin,297.17,106.15,0.00),v40,z0,tPen\WObj:=wPaper;
    MoveL Offs(pOrigin,297.60,105.51,0.00),v40,z0,tPen\WObj:=wPaper;
    MoveL Offs(pOrigin,318.21,110.40,0.00),v40,z0,tPen\WObj:=wPaper;
    MoveL Offs(pOrigin,339.46,116.35,0.00),v40,z0,tPen\WObj:=wPaper;
    MoveL Offs(pOrigin,344.35,117.98,0.00),v40,z0,tPen\WObj:=wPaper;
  ENDPROC

  PROC DrawPart70()
    MoveL Offs(pOrigin,345.34,118.69,0.00),v40,z0,tPen\WObj:=wPaper;
    MoveL Offs(pOrigin,345.62,119.32,0.00),v40,z0,tPen\WObj:=wPaper;
    MoveL Offs(pOrigin,345.84,124.85,0.00),v40,z0,tPen\WObj:=wPaper;
    MoveL Offs(pOrigin,345.62,128.46,0.00),v40,z0,tPen\WObj:=wPaper;
    MoveL Offs(pOrigin,345.20,130.09,0.00),v40,z0,tPen\WObj:=wPaper;
    MoveL Offs(pOrigin,344.56,130.38,0.00),v40,z0,tPen\WObj:=wPaper;
    MoveL Offs(pOrigin,336.06,127.82,0.00),v40,z0,tPen\WObj:=wPaper;
    MoveL Offs(pOrigin,335.00,128.04,0.00),v40,z0,tPen\WObj:=wPaper;
    MoveL Offs(pOrigin,335.00,128.04,0.00),v40,z0,tPen\WObj:=wPaper;
    MoveL Offs(pOrigin,335.21,128.68,0.00),v40,z0,tPen\WObj:=wPaper;
    MoveL Offs(pOrigin,339.89,132.71,0.00),v40,z0,tPen\WObj:=wPaper;
    MoveL Offs(pOrigin,348.39,138.45,0.00),v40,fine,tPen\WObj:=wPaper;
    MoveL Offs(pOrigin,348.39,138.45,6.00),v60,z5,tPen\WObj:=wPaper;
    MoveL Offs(pOrigin,347.10,137.01,6.00),vTravel,z5,tPen\WObj:=wPaper;
    MoveL Offs(pOrigin,347.10,137.01,0.00),v60,z0,tPen\WObj:=wPaper;
    MoveL Offs(pOrigin,346.20,137.92,0.00),v40,z0,tPen\WObj:=wPaper;
    MoveL Offs(pOrigin,345.30,137.32,0.00),v40,z0,tPen\WObj:=wPaper;
    MoveL Offs(pOrigin,346.20,136.42,0.00),v40,z0,tPen\WObj:=wPaper;
    MoveL Offs(pOrigin,345.30,135.82,0.00),v40,z0,tPen\WObj:=wPaper;
    MoveL Offs(pOrigin,344.25,136.87,0.00),v40,z0,tPen\WObj:=wPaper;
    MoveL Offs(pOrigin,343.36,136.28,0.00),v40,z0,tPen\WObj:=wPaper;
    MoveL Offs(pOrigin,344.71,134.93,0.00),v40,z0,tPen\WObj:=wPaper;
    MoveL Offs(pOrigin,343.81,134.33,0.00),v40,z0,tPen\WObj:=wPaper;
    MoveL Offs(pOrigin,342.31,135.83,0.00),v40,z0,tPen\WObj:=wPaper;
    MoveL Offs(pOrigin,342.22,134.92,0.00),v40,z0,tPen\WObj:=wPaper;
    MoveL Offs(pOrigin,332.75,125.46,0.00),v40,fine,tPen\WObj:=wPaper;
    MoveL Offs(pOrigin,332.75,125.46,6.00),v60,z5,tPen\WObj:=wPaper;
    MoveL Offs(pOrigin,332.89,124.11,6.00),vTravel,z5,tPen\WObj:=wPaper;
    MoveL Offs(pOrigin,332.89,124.11,0.00),v60,z0,tPen\WObj:=wPaper;
    MoveL Offs(pOrigin,331.69,122.91,0.00),v40,z0,tPen\WObj:=wPaper;
    MoveL Offs(pOrigin,332.01,122.23,0.00),v40,z0,tPen\WObj:=wPaper;
    MoveL Offs(pOrigin,327.96,126.29,0.00),v40,z0,tPen\WObj:=wPaper;
    MoveL Offs(pOrigin,329.01,126.20,0.00),v40,z0,tPen\WObj:=wPaper;
    MoveL Offs(pOrigin,326.45,123.64,0.00),v40,fine,tPen\WObj:=wPaper;
    MoveL Offs(pOrigin,326.45,123.64,6.00),v60,z5,tPen\WObj:=wPaper;
    MoveL Offs(pOrigin,326.60,122.29,6.00),vTravel,z5,tPen\WObj:=wPaper;
    MoveL Offs(pOrigin,326.60,122.29,0.00),v60,z0,tPen\WObj:=wPaper;
    MoveL Offs(pOrigin,325.70,121.39,0.00),v40,z0,tPen\WObj:=wPaper;
    MoveL Offs(pOrigin,326.03,120.75,0.00),v40,z0,tPen\WObj:=wPaper;
    MoveL Offs(pOrigin,322.12,124.66,0.00),v40,z0,tPen\WObj:=wPaper;
    MoveL Offs(pOrigin,322.56,124.23,0.00),v40,z0,tPen\WObj:=wPaper;
    MoveL Offs(pOrigin,320.15,121.82,0.00),v40,fine,tPen\WObj:=wPaper;
    MoveL Offs(pOrigin,320.15,121.82,6.00),v60,z5,tPen\WObj:=wPaper;
    MoveL Offs(pOrigin,320.46,123.62,6.00),vTravel,z5,tPen\WObj:=wPaper;
    MoveL Offs(pOrigin,320.46,123.62,0.00),v60,z0,tPen\WObj:=wPaper;
    MoveL Offs(pOrigin,318.06,121.22,0.00),v40,fine,tPen\WObj:=wPaper;
    MoveL Offs(pOrigin,318.06,121.22,6.00),v60,z5,tPen\WObj:=wPaper;
    MoveL Offs(pOrigin,318.51,123.17,6.00),vTravel,z5,tPen\WObj:=wPaper;
    MoveL Offs(pOrigin,318.51,123.17,0.00),v60,z0,tPen\WObj:=wPaper;
    MoveL Offs(pOrigin,316.11,120.76,0.00),v40,fine,tPen\WObj:=wPaper;
    MoveL Offs(pOrigin,316.11,120.76,6.00),v60,z5,tPen\WObj:=wPaper;
    MoveL Offs(pOrigin,316.41,122.56,6.00),vTravel,z5,tPen\WObj:=wPaper;
    MoveL Offs(pOrigin,316.41,122.56,0.00),v60,z0,tPen\WObj:=wPaper;
    MoveL Offs(pOrigin,314.01,120.16,0.00),v40,fine,tPen\WObj:=wPaper;
    MoveL Offs(pOrigin,314.01,120.16,6.00),v60,z5,tPen\WObj:=wPaper;
    MoveL Offs(pOrigin,312.21,119.85,6.00),vTravel,z5,tPen\WObj:=wPaper;
    MoveL Offs(pOrigin,312.21,119.85,0.00),v60,z0,tPen\WObj:=wPaper;
    MoveL Offs(pOrigin,314.61,122.26,0.00),v40,z0,tPen\WObj:=wPaper;
    MoveL Offs(pOrigin,314.04,122.29,0.00),v40,z0,tPen\WObj:=wPaper;
    MoveL Offs(pOrigin,317.79,118.53,0.00),v40,fine,tPen\WObj:=wPaper;
    MoveL Offs(pOrigin,317.79,118.53,6.00),v60,z5,tPen\WObj:=wPaper;
    MoveL Offs(pOrigin,319.14,118.68,6.00),vTravel,z5,tPen\WObj:=wPaper;
    MoveL Offs(pOrigin,319.14,118.68,0.00),v60,z0,tPen\WObj:=wPaper;
    MoveL Offs(pOrigin,315.24,122.58,0.00),v40,z0,tPen\WObj:=wPaper;
    MoveL Offs(pOrigin,316.28,123.03,0.00),v40,z0,tPen\WObj:=wPaper;
    MoveL Offs(pOrigin,320.19,119.12,0.00),v40,fine,tPen\WObj:=wPaper;
    MoveL Offs(pOrigin,320.19,119.12,6.00),v60,z5,tPen\WObj:=wPaper;
    MoveL Offs(pOrigin,321.39,119.42,6.00),vTravel,z5,tPen\WObj:=wPaper;
    MoveL Offs(pOrigin,321.39,119.42,0.00),v60,z0,tPen\WObj:=wPaper;
    MoveL Offs(pOrigin,317.48,123.32,0.00),v40,fine,tPen\WObj:=wPaper;
    MoveL Offs(pOrigin,317.48,123.32,6.00),v60,z5,tPen\WObj:=wPaper;
    MoveL Offs(pOrigin,318.68,123.62,6.00),vTravel,z5,tPen\WObj:=wPaper;
    MoveL Offs(pOrigin,318.68,123.62,0.00),v60,z0,tPen\WObj:=wPaper;
    MoveL Offs(pOrigin,322.58,119.71,0.00),v40,fine,tPen\WObj:=wPaper;
    MoveL Offs(pOrigin,322.58,119.71,6.00),v60,z5,tPen\WObj:=wPaper;
    MoveL Offs(pOrigin,323.78,120.01,6.00),vTravel,z5,tPen\WObj:=wPaper;
    MoveL Offs(pOrigin,323.78,120.01,0.00),v60,z0,tPen\WObj:=wPaper;
    MoveL Offs(pOrigin,319.88,123.92,0.00),v40,fine,tPen\WObj:=wPaper;
    MoveL Offs(pOrigin,319.88,123.92,6.00),v60,z5,tPen\WObj:=wPaper;
    MoveL Offs(pOrigin,321.07,124.21,6.00),vTravel,z5,tPen\WObj:=wPaper;
    MoveL Offs(pOrigin,321.07,124.21,0.00),v60,z0,tPen\WObj:=wPaper;
    MoveL Offs(pOrigin,324.83,120.46,0.00),v40,fine,tPen\WObj:=wPaper;
    MoveL Offs(pOrigin,324.83,120.46,6.00),v60,z5,tPen\WObj:=wPaper;
    MoveL Offs(pOrigin,327.22,121.05,6.00),vTravel,z5,tPen\WObj:=wPaper;
    MoveL Offs(pOrigin,327.22,121.05,0.00),v60,z0,tPen\WObj:=wPaper;
    MoveL Offs(pOrigin,323.32,124.95,0.00),v40,fine,tPen\WObj:=wPaper;
    MoveL Offs(pOrigin,323.32,124.95,6.00),v60,z5,tPen\WObj:=wPaper;
    MoveL Offs(pOrigin,324.52,125.25,6.00),vTravel,z5,tPen\WObj:=wPaper;
    MoveL Offs(pOrigin,324.52,125.25,0.00),v60,z0,tPen\WObj:=wPaper;
    MoveL Offs(pOrigin,328.42,121.34,0.00),v40,z0,tPen\WObj:=wPaper;
    MoveL Offs(pOrigin,327.64,121.85,0.00),v40,z0,tPen\WObj:=wPaper;
    MoveL Offs(pOrigin,328.85,123.05,0.00),v40,z0,tPen\WObj:=wPaper;
    MoveL Offs(pOrigin,329.74,122.45,0.00),v40,z0,tPen\WObj:=wPaper;
    MoveL Offs(pOrigin,330.95,123.66,0.00),v40,fine,tPen\WObj:=wPaper;
    MoveL Offs(pOrigin,330.95,123.66,6.00),v60,z5,tPen\WObj:=wPaper;
    MoveL Offs(pOrigin,330.65,124.85,6.00),vTravel,z5,tPen\WObj:=wPaper;
    MoveL Offs(pOrigin,330.65,124.85,0.00),v60,z0,tPen\WObj:=wPaper;
    MoveL Offs(pOrigin,335.61,129.81,0.00),v40,z0,tPen\WObj:=wPaper;
    MoveL Offs(pOrigin,334.84,129.86,0.00),v40,z0,tPen\WObj:=wPaper;
    MoveL Offs(pOrigin,340.10,124.60,0.00),v40,z0,tPen\WObj:=wPaper;
    MoveL Offs(pOrigin,341.14,125.05,0.00),v40,z0,tPen\WObj:=wPaper;
    MoveL Offs(pOrigin,335.58,130.61,0.00),v40,z0,tPen\WObj:=wPaper;
    MoveL Offs(pOrigin,336.48,131.21,0.00),v40,z0,tPen\WObj:=wPaper;
    MoveL Offs(pOrigin,341.89,125.80,0.00),v40,z0,tPen\WObj:=wPaper;
    MoveL Offs(pOrigin,342.23,126.34,0.00),v40,z0,tPen\WObj:=wPaper;
    MoveL Offs(pOrigin,333.73,123.79,0.00),v40,z0,tPen\WObj:=wPaper;
    MoveL Offs(pOrigin,300.15,114.86,0.00),v40,z0,tPen\WObj:=wPaper;
    MoveL Offs(pOrigin,299.98,115.44,0.00),v40,z0,tPen\WObj:=wPaper;
    MoveL Offs(pOrigin,296.22,119.20,0.00),v40,z0,tPen\WObj:=wPaper;
    MoveL Offs(pOrigin,296.63,119.21,0.00),v40,z0,tPen\WObj:=wPaper;
    MoveL Offs(pOrigin,300.08,122.66,0.00),v40,z0,tPen\WObj:=wPaper;
    MoveL Offs(pOrigin,299.73,122.71,0.00),v40,z0,tPen\WObj:=wPaper;
    MoveL Offs(pOrigin,298.45,122.71,0.00),v40,z0,tPen\WObj:=wPaper;
    MoveL Offs(pOrigin,298.14,123.70,0.00),v40,z0,tPen\WObj:=wPaper;
    MoveL Offs(pOrigin,301.30,126.86,0.00),v40,z0,tPen\WObj:=wPaper;
    MoveL Offs(pOrigin,301.00,126.94,0.00),v40,z0,tPen\WObj:=wPaper;
    MoveL Offs(pOrigin,299.94,126.94,0.00),v40,z0,tPen\WObj:=wPaper;
    MoveL Offs(pOrigin,300.15,127.99,0.00),v40,z0,tPen\WObj:=wPaper;
    MoveL Offs(pOrigin,301.21,127.99,0.00),v40,z0,tPen\WObj:=wPaper;
    MoveL Offs(pOrigin,302.19,128.16,0.00),v40,z0,tPen\WObj:=wPaper;
  ENDPROC

  PROC DrawPart71()
    MoveL Offs(pOrigin,299.78,130.57,0.00),v40,z0,tPen\WObj:=wPaper;
    MoveL Offs(pOrigin,300.26,130.30,0.00),v40,z0,tPen\WObj:=wPaper;
    MoveL Offs(pOrigin,303.56,133.61,0.00),v40,z0,tPen\WObj:=wPaper;
    MoveL Offs(pOrigin,304.12,133.70,0.00),v40,z0,tPen\WObj:=wPaper;
    MoveL Offs(pOrigin,301.56,136.26,0.00),v40,z0,tPen\WObj:=wPaper;
    MoveL Offs(pOrigin,302.38,136.90,0.00),v40,z0,tPen\WObj:=wPaper;
    MoveL Offs(pOrigin,305.68,140.21,0.00),v40,z0,tPen\WObj:=wPaper;
    MoveL Offs(pOrigin,305.25,140.66,0.00),v40,z0,tPen\WObj:=wPaper;
    MoveL Offs(pOrigin,304.19,140.66,0.00),v40,z0,tPen\WObj:=wPaper;
    MoveL Offs(pOrigin,303.44,140.95,0.00),v40,z0,tPen\WObj:=wPaper;
    MoveL Offs(pOrigin,306.89,144.40,0.00),v40,z0,tPen\WObj:=wPaper;
    MoveL Offs(pOrigin,306.52,144.89,0.00),v40,z0,tPen\WObj:=wPaper;
    MoveL Offs(pOrigin,305.46,144.89,0.00),v40,z0,tPen\WObj:=wPaper;
    MoveL Offs(pOrigin,304.95,145.45,0.00),v40,z0,tPen\WObj:=wPaper;
    MoveL Offs(pOrigin,308.25,148.75,0.00),v40,z0,tPen\WObj:=wPaper;
    MoveL Offs(pOrigin,308.71,148.52,0.00),v40,z0,tPen\WObj:=wPaper;
    MoveL Offs(pOrigin,306.31,150.92,0.00),v40,z0,tPen\WObj:=wPaper;
    MoveL Offs(pOrigin,306.46,149.94,0.00),v40,z0,tPen\WObj:=wPaper;
    MoveL Offs(pOrigin,309.77,153.25,0.00),v40,fine,tPen\WObj:=wPaper;
    MoveL Offs(pOrigin,309.77,153.25,6.00),v60,z5,tPen\WObj:=wPaper;
    MoveL Offs(pOrigin,309.46,150.76,6.00),vTravel,z5,tPen\WObj:=wPaper;
    MoveL Offs(pOrigin,309.46,150.76,0.00),v60,z0,tPen\WObj:=wPaper;
    MoveL Offs(pOrigin,306.90,153.32,0.00),v40,fine,tPen\WObj:=wPaper;
    MoveL Offs(pOrigin,306.90,153.32,6.00),v60,z5,tPen\WObj:=wPaper;
    MoveL Offs(pOrigin,306.61,152.12,6.00),vTravel,z5,tPen\WObj:=wPaper;
    MoveL Offs(pOrigin,306.61,152.12,0.00),v60,z0,tPen\WObj:=wPaper;
    MoveL Offs(pOrigin,309.01,149.71,0.00),v40,z0,tPen\WObj:=wPaper;
    MoveL Offs(pOrigin,308.23,150.17,0.00),v40,z0,tPen\WObj:=wPaper;
    MoveL Offs(pOrigin,307.16,150.17,0.00),v40,fine,tPen\WObj:=wPaper;
    MoveL Offs(pOrigin,307.16,150.17,6.00),v60,z5,tPen\WObj:=wPaper;
    MoveL Offs(pOrigin,305.86,149.87,6.00),vTravel,z5,tPen\WObj:=wPaper;
    MoveL Offs(pOrigin,305.86,149.87,0.00),v60,z0,tPen\WObj:=wPaper;
    MoveL Offs(pOrigin,308.42,147.32,0.00),v40,z0,tPen\WObj:=wPaper;
    MoveL Offs(pOrigin,307.59,148.06,0.00),v40,z0,tPen\WObj:=wPaper;
    MoveL Offs(pOrigin,306.52,148.06,0.00),v40,z0,tPen\WObj:=wPaper;
    MoveL Offs(pOrigin,305.55,147.55,0.00),v40,z0,tPen\WObj:=wPaper;
    MoveL Offs(pOrigin,308.86,150.85,0.00),v40,fine,tPen\WObj:=wPaper;
    MoveL Offs(pOrigin,308.86,150.85,6.00),v60,z5,tPen\WObj:=wPaper;
    MoveL Offs(pOrigin,305.57,148.68,6.00),vTravel,z5,tPen\WObj:=wPaper;
    MoveL Offs(pOrigin,305.57,148.68,0.00),v60,z0,tPen\WObj:=wPaper;
    MoveL Offs(pOrigin,307.97,146.27,0.00),v40,z0,tPen\WObj:=wPaper;
    MoveL Offs(pOrigin,307.50,146.50,0.00),v40,z0,tPen\WObj:=wPaper;
    MoveL Offs(pOrigin,304.34,143.35,0.00),v40,z0,tPen\WObj:=wPaper;
    MoveL Offs(pOrigin,303.79,142.99,0.00),v40,z0,tPen\WObj:=wPaper;
    MoveL Offs(pOrigin,306.34,140.44,0.00),v40,z0,tPen\WObj:=wPaper;
    MoveL Offs(pOrigin,305.90,139.39,0.00),v40,z0,tPen\WObj:=wPaper;
    MoveL Offs(pOrigin,303.34,141.94,0.00),v40,z0,tPen\WObj:=wPaper;
    MoveL Offs(pOrigin,302.90,140.90,0.00),v40,z0,tPen\WObj:=wPaper;
    MoveL Offs(pOrigin,305.45,138.34,0.00),v40,z0,tPen\WObj:=wPaper;
    MoveL Offs(pOrigin,304.77,137.81,0.00),v40,z0,tPen\WObj:=wPaper;
    MoveL Offs(pOrigin,301.47,134.50,0.00),v40,z0,tPen\WObj:=wPaper;
    MoveL Offs(pOrigin,301.27,135.06,0.00),v40,z0,tPen\WObj:=wPaper;
    MoveL Offs(pOrigin,303.67,132.65,0.00),v40,z0,tPen\WObj:=wPaper;
    MoveL Offs(pOrigin,302.91,133.27,0.00),v40,z0,tPen\WObj:=wPaper;
    MoveL Offs(pOrigin,301.85,133.27,0.00),v40,z0,tPen\WObj:=wPaper;
    MoveL Offs(pOrigin,302.27,134.33,0.00),v40,z0,tPen\WObj:=wPaper;
    MoveL Offs(pOrigin,303.34,134.33,0.00),v40,z0,tPen\WObj:=wPaper;
    MoveL Offs(pOrigin,303.55,135.38,0.00),v40,z0,tPen\WObj:=wPaper;
    MoveL Offs(pOrigin,302.49,135.38,0.00),v40,z0,tPen\WObj:=wPaper;
    MoveL Offs(pOrigin,302.91,136.44,0.00),v40,z0,tPen\WObj:=wPaper;
    MoveL Offs(pOrigin,303.98,136.44,0.00),v40,z0,tPen\WObj:=wPaper;
    MoveL Offs(pOrigin,304.17,135.71,0.00),v40,z0,tPen\WObj:=wPaper;
    MoveL Offs(pOrigin,300.86,132.40,0.00),v40,z0,tPen\WObj:=wPaper;
    MoveL Offs(pOrigin,300.52,132.81,0.00),v40,z0,tPen\WObj:=wPaper;
    MoveL Offs(pOrigin,303.08,130.26,0.00),v40,z0,tPen\WObj:=wPaper;
    MoveL Offs(pOrigin,302.06,130.10,0.00),v40,z0,tPen\WObj:=wPaper;
    MoveL Offs(pOrigin,300.79,130.10,0.00),v40,z0,tPen\WObj:=wPaper;
    MoveL Offs(pOrigin,300.58,129.05,0.00),v40,z0,tPen\WObj:=wPaper;
    MoveL Offs(pOrigin,301.64,129.05,0.00),v40,z0,tPen\WObj:=wPaper;
    MoveL Offs(pOrigin,302.20,129.26,0.00),v40,z0,tPen\WObj:=wPaper;
    MoveL Offs(pOrigin,298.75,125.80,0.00),v40,z0,tPen\WObj:=wPaper;
    MoveL Offs(pOrigin,298.30,126.08,0.00),v40,z0,tPen\WObj:=wPaper;
    MoveL Offs(pOrigin,301.00,123.37,0.00),v40,z0,tPen\WObj:=wPaper;
    MoveL Offs(pOrigin,299.94,123.77,0.00),v40,z0,tPen\WObj:=wPaper;
    MoveL Offs(pOrigin,298.88,123.77,0.00),v40,z0,tPen\WObj:=wPaper;
    MoveL Offs(pOrigin,299.09,124.82,0.00),v40,z0,tPen\WObj:=wPaper;
    MoveL Offs(pOrigin,300.36,124.82,0.00),v40,z0,tPen\WObj:=wPaper;
    MoveL Offs(pOrigin,300.99,125.06,0.00),v40,z0,tPen\WObj:=wPaper;
    MoveL Offs(pOrigin,297.23,121.30,0.00),v40,z0,tPen\WObj:=wPaper;
    MoveL Offs(pOrigin,296.96,121.44,0.00),v40,z0,tPen\WObj:=wPaper;
    MoveL Offs(pOrigin,303.27,115.13,0.00),v40,fine,tPen\WObj:=wPaper;
    MoveL Offs(pOrigin,303.27,115.13,6.00),v60,z5,tPen\WObj:=wPaper;
    MoveL Offs(pOrigin,304.47,115.42,6.00),vTravel,z5,tPen\WObj:=wPaper;
    MoveL Offs(pOrigin,304.47,115.42,0.00),v60,z0,tPen\WObj:=wPaper;
    MoveL Offs(pOrigin,301.17,118.73,0.00),v40,z0,tPen\WObj:=wPaper;
    MoveL Offs(pOrigin,302.02,118.62,0.00),v40,z0,tPen\WObj:=wPaper;
    MoveL Offs(pOrigin,299.77,116.37,0.00),v40,z0,tPen\WObj:=wPaper;
    MoveL Offs(pOrigin,298.88,116.38,0.00),v40,z0,tPen\WObj:=wPaper;
    MoveL Offs(pOrigin,296.54,116.38,0.00),v40,z0,tPen\WObj:=wPaper;
    MoveL Offs(pOrigin,296.02,117.11,0.00),v40,z0,tPen\WObj:=wPaper;
    MoveL Offs(pOrigin,299.48,120.56,0.00),v40,z0,tPen\WObj:=wPaper;
    MoveL Offs(pOrigin,299.81,120.08,0.00),v40,z0,tPen\WObj:=wPaper;
    MoveL Offs(pOrigin,297.26,122.64,0.00),v40,z0,tPen\WObj:=wPaper;
    MoveL Offs(pOrigin,297.71,123.68,0.00),v40,z0,tPen\WObj:=wPaper;
    MoveL Offs(pOrigin,300.11,121.28,0.00),v40,z0,tPen\WObj:=wPaper;
    MoveL Offs(pOrigin,299.30,121.66,0.00),v40,z0,tPen\WObj:=wPaper;
    MoveL Offs(pOrigin,298.24,121.66,0.00),v40,z0,tPen\WObj:=wPaper;
    MoveL Offs(pOrigin,297.81,120.60,0.00),v40,z0,tPen\WObj:=wPaper;
    MoveL Offs(pOrigin,298.88,120.60,0.00),v40,z0,tPen\WObj:=wPaper;
    MoveL Offs(pOrigin,298.66,119.54,0.00),v40,z0,tPen\WObj:=wPaper;
    MoveL Offs(pOrigin,297.60,119.54,0.00),v40,z0,tPen\WObj:=wPaper;
    MoveL Offs(pOrigin,297.18,118.49,0.00),v40,z0,tPen\WObj:=wPaper;
    MoveL Offs(pOrigin,298.45,118.49,0.00),v40,z0,tPen\WObj:=wPaper;
    MoveL Offs(pOrigin,299.02,118.61,0.00),v40,z0,tPen\WObj:=wPaper;
    MoveL Offs(pOrigin,295.27,114.86,0.00),v40,z0,tPen\WObj:=wPaper;
    MoveL Offs(pOrigin,294.74,114.71,0.00),v40,z0,tPen\WObj:=wPaper;
    MoveL Offs(pOrigin,297.44,112.00,0.00),v40,z0,tPen\WObj:=wPaper;
    MoveL Offs(pOrigin,296.61,111.72,0.00),v40,z0,tPen\WObj:=wPaper;
    MoveL Offs(pOrigin,293.15,108.26,0.00),v40,z0,tPen\WObj:=wPaper;
    MoveL Offs(pOrigin,293.11,108.87,0.00),v40,z0,tPen\WObj:=wPaper;
    MoveL Offs(pOrigin,297.31,104.66,0.00),v40,z0,tPen\WObj:=wPaper;
    MoveL Offs(pOrigin,297.17,105.51,0.00),v40,z0,tPen\WObj:=wPaper;
    MoveL Offs(pOrigin,296.11,105.30,0.00),v40,z0,tPen\WObj:=wPaper;
    MoveL Offs(pOrigin,296.11,105.30,0.00),v40,z0,tPen\WObj:=wPaper;
    MoveL Offs(pOrigin,294.27,104.88,0.00),v40,z0,tPen\WObj:=wPaper;
    MoveL Offs(pOrigin,293.14,100.84,0.00),v40,z0,tPen\WObj:=wPaper;
    MoveL Offs(pOrigin,292.29,96.59,0.00),v40,z0,tPen\WObj:=wPaper;
    MoveL Offs(pOrigin,291.86,82.78,0.00),v40,z0,tPen\WObj:=wPaper;
    MoveL Offs(pOrigin,292.50,75.34,0.00),v40,z0,tPen\WObj:=wPaper;
    MoveL Offs(pOrigin,293.77,67.90,0.00),v40,z0,tPen\WObj:=wPaper;
  ENDPROC

